// TwinCAT 3 PLC project PLC1
// Title: TcHAL
// Company: none
// Author: Tobias Freyermuth
// ProjectVersion: 0.1.4
// Description: Hardware Abstraction Layer of TwinCAT fieldbus devices
// ProgramVersion: 3.1.4024.12
// libraries:
//   Tc2_EtherCAT, * (Beckhoff Automation GmbH)
//   Tc2_Standard, * (Beckhoff Automation GmbH)
//   Tc2_System, * (Beckhoff Automation GmbH)
//   Tc3_Module, * (Beckhoff Automation GmbH)
//   TcUnit, * (www.tcunit.org)
// project tree:
//   analog_input/temperature/ EL3202_0010.TcPOU
//   analog_input/voltage/ EL3164.TcPOU
//   analog_input/_internal/ AI_Voltage_Channel.TcPOU, AI_Temperature_Channel.TcPOU, I_AI_percentage.TcIO, I_AI_Temperature.TcIO, I_AI_Voltage.TcIO
//   analog_output/voltage/ EL4002.TcPOU, EL4102.TcPOU, EL4004.TcPOU, EL4134.TcPOU
//   analog_output/_internal/ AO_Voltage_Channel.TcPOU, I_AO_percentage.TcIO, I_AO_Voltage.TcIO
//   coupler/ EK1101.TcPOU
//   digital_input/ EL1008.TcPOU, EL1104.TcPOU, EL1144.TcPOU, EL1808.TcPOU, EL1124.TcPOU, EL1809.TcPOU
//   digital_input/_internal/ HAL_DI_Channel.TcPOU, I_HAL_DI.TcIO
//   digital_output/ EL2008.TcPOU, EL2124.TcPOU, EL2024_0010.TcPOU, EL2502.TcPOU (excluded from build), EL2595.TcPOU, EL2612.TcPOU, EL2521.TcPOU (excluded from build), EL2004.TcPOU, EL2634.TcPOU, EL2808.TcPOU, EL2624.TcPOU, EL2794.TcPOU
//   digital_output/_internal/ HAL_DO_Channel.TcPOU, I_HAL_DO.TcIO
//   / HAL_ErrorEnum.TcDUT, MAIN.TcPOU, PlcTask.TcTTO, Settings.TcGVL, _internal.TcGVL
//   InterfaceManager/ InterfaceManager.TcPOU, InterfaceManager_test.TcPOU, I_AI_Percentage_register.TcDUT, I_AO_Percentage_register.TcDUT, I_AO_Voltage_register.TcDUT, I_AI_Voltage_register.TcDUT, I_InterfaceManager.TcIO
//   Project Information/ F_GetCompany.TcPOU, F_GetTitle.TcPOU (not stored), F_GetVersion.TcPOU
//   Version/ Global_Version.TcGVL
//   _internal/CoE/BeckhoffTerminalConfigEnums/ ENU_DT0800EN02.TcDUT (not stored), ENU_DT0801EN03.TcDUT (not stored)
//   _internal/CoE/buffer/ ring_buffer_CoE_read.TcPOU
//   _internal/CoE/ CoE_buffer_type_cast_union.TcDUT (not stored), CoE_communication_handler.TcPOU, CoE_property_handler.TcPOU, CoE_UML_Class Diagram.TcCD (not stored), I_CoE_config_common.TcIO, I_CoE_property.TcIO, I_CoE_communication_handler.TcIO
//   _internal/CoE/properties/ CoE_property.TcPOU, CoE_property_bool.TcPOU, CoE_property_dint.TcPOU, CoE_property_int.TcPOU, CoE_property_string.TcPOU, CoE_property_udint.TcPOU, CoE_property_uint.TcPOU, CoE_property_usint.TcPOU
//   _internal/ I_device_control.TcIO, I_terminal_channel.TcIO, I_coupler_execution.TcIO, I_terminal_execution.TcIO, linear_adc_to_phy.TcPOU, linear_phy_to_adc.TcPOU, linear_phy_to_adc_test.TcPOU, linear_adc_to_phy_test.TcPOU
// real-time tasks:
//   TASK PlcTask: cycle T#10ms, priority 20, ADS port 350

CONFIGURATION PLC1
    RESOURCE PLC ON TwinCAT3
        TASK PlcTask(INTERVAL := T#10ms, PRIORITY := 20);
        PROGRAM MAIN WITH PlcTask : MAIN;
    END_RESOURCE
END_CONFIGURATION

// ---- HAL_ErrorEnum.TcDUT
(**
This error enum is the central error return type used accross all POUs within TcHAL.
*)

{attribute 'qualified_only'}
{attribute 'strict'}
TYPE HAL_ErrorEnum :
(
	no_error := 0,
	// Error messages related to InterfaceManager
	terminal_not_found, 
	interface_can_not_be_null,
	terminal_name_can_not_be_empty,
	channel_number_out_of_range,
	device_id_can_not_be_null,
	no_empty_space_found_in_register,
	requested_interface_not_found,
	interface_already_in_use,
	max_registration_limit_per_cycle_reached,
    physical_value_too_big,
    physical_value_too_small,
    dx_zero_or_smaller,
    m_zero_or_smaller
);
END_TYPE

// ---- InterfaceManager/I_AI_Percentage_register.TcDUT
TYPE I_AI_Percentage_register :
STRUCT
	registered_interface			: I_AI_Percentage;
	terminal_id 					: UINT;
	channel_number 					: USINT;
	connected_device_id				: UINT;
END_STRUCT
END_TYPE

// ---- InterfaceManager/I_AO_Percentage_register.TcDUT
TYPE I_AO_Percentage_register :
STRUCT
	registered_interface			: I_AO_Percentage;
	terminal_id 					: UINT;
	channel_number 					: USINT;
	connected_device_id				: UINT;
END_STRUCT
END_TYPE

// ---- InterfaceManager/I_AO_Voltage_register.TcDUT
TYPE I_AO_Voltage_register :
STRUCT
	registered_interface			: I_AO_Voltage;
	terminal_id 					: UINT;
	channel_number 					: USINT;
	connected_device_id				: UINT;
END_STRUCT
END_TYPE

// ---- InterfaceManager/I_AI_Voltage_register.TcDUT
TYPE I_AI_Voltage_register :
STRUCT
	registered_interface			: I_AI_Voltage;
	terminal_id 					: UINT;
	channel_number 					: USINT;
	connected_device_id				: UINT;
END_STRUCT
END_TYPE

// ---- Settings.TcGVL
VAR_GLOBAL CONSTANT
	NUMBER_OF_TERMINALS 	: UINT:=200;

	NUMBER_OF_I_HAL_AO_Voltage_INTERFACES		: UINT:=10;
	NUMBER_OF_I_HAL_AI_Voltage_INTERFACES		: UINT:=10;
	NUMBER_OF_I_AI_Percentage_INTERFACES		: UINT:=10;

END_VAR

// ---- Version/Global_Version.TcGVL
{attribute 'TcGenerated'}
{attribute 'no-analysis'}
{attribute 'linkalways'}
// This function has been automatically generated from the project information.
VAR_GLOBAL CONSTANT
	{attribute 'const_non_replaced'}
	stLibVersion_TcHAL : ST_LibVersion := (iMajor := 0, iMinor := 1, iBuild := 4, iRevision := 0, nFlags := 0, sVersion := '0.1.4');
END_VAR

// ---- _internal.TcGVL
{attribute 'qualified_only'}
VAR_GLOBAL
	InterfaceManager_InstanceCounter :UINT;
END_VAR

// ---- analog_input/_internal/I_AI_percentage.TcIO
INTERFACE I_AI_percentage

PROPERTY max_value : real
GET
END_GET
SET
END_SET
END_PROPERTY

PROPERTY min_value : real
GET
END_GET
SET
END_SET
END_PROPERTY

PROPERTY value : real
GET
END_GET
END_PROPERTY

END_INTERFACE

// ---- analog_input/_internal/I_AI_Temperature.TcIO
INTERFACE I_AI_Temperature

PROPERTY errId : HAL_ErrorEnum
GET
END_GET
END_PROPERTY

PROPERTY value : real
GET
END_GET
END_PROPERTY

END_INTERFACE

// ---- analog_input/_internal/I_AI_Voltage.TcIO
INTERFACE I_AI_Voltage

PROPERTY errId : HAL_ErrorEnum
GET
END_GET
END_PROPERTY

PROPERTY rValue : real
GET
END_GET
END_PROPERTY

END_INTERFACE

// ---- analog_output/_internal/I_AO_percentage.TcIO
INTERFACE I_AO_percentage

PROPERTY max_value : real
GET
END_GET
SET
END_SET
END_PROPERTY

PROPERTY min_value : real
GET
END_GET
SET
END_SET
END_PROPERTY

PROPERTY value : real
GET
END_GET
END_PROPERTY

END_INTERFACE

// ---- analog_output/_internal/I_AO_Voltage.TcIO
INTERFACE I_AO_Voltage

PROPERTY errId : HAL_ErrorEnum
GET
END_GET
END_PROPERTY

PROPERTY rValue : real
GET
END_GET
SET
END_SET
END_PROPERTY

END_INTERFACE

// ---- digital_input/_internal/I_HAL_DI.TcIO
INTERFACE I_HAL_DI

PROPERTY errId : uint
GET
END_GET
END_PROPERTY

PROPERTY xValue : bool
GET
END_GET
END_PROPERTY

END_INTERFACE

// ---- digital_output/_internal/I_HAL_DO.TcIO
INTERFACE I_HAL_DO

PROPERTY errId : HAL_ErrorEnum
GET
END_GET
END_PROPERTY

PROPERTY xValue : bool
GET
END_GET
SET
END_SET
END_PROPERTY

END_INTERFACE

// ---- InterfaceManager/I_InterfaceManager.TcIO
INTERFACE I_InterfaceManager

METHOD register_I_AI_Percentage : BOOL
VAR_INPUT
	interface_to_be_registered		: I_AI_Percentage;
	terminal_id 					: UINT;
	channel_number 					: USINT; 
END_VAR
VAR_OUTPUT
	errId		: HAL_ErrorEnum;
END_VAR
END_METHOD

METHOD register_I_AI_Temperature : BOOL
VAR_INPUT
	interface_to_be_registered		: I_AI_Temperature;
	terminal_id 					: UINT;
	channel_number 					: USINT; 
END_VAR
VAR_OUTPUT
	errId		: HAL_ErrorEnum;
END_VAR
END_METHOD

METHOD register_I_AI_Voltage : BOOL
VAR_INPUT
	interface_to_be_registered		: I_AI_Voltage;
	terminal_id 					: UINT;
	channel_number 					: USINT; 
END_VAR
VAR_OUTPUT
	errId		: HAL_ErrorEnum;
END_VAR
END_METHOD

METHOD register_I_AO_Percentage : BOOL
VAR_INPUT
	interface_to_be_registered		: I_AO_Percentage;
	terminal_id 					: UINT;
	channel_number 					: USINT; 
END_VAR
VAR_OUTPUT
	errId		: HAL_ErrorEnum;
END_VAR
END_METHOD

METHOD register_I_AO_Voltage : BOOL
VAR_INPUT
	interface_to_be_registered		: I_AO_Voltage;
	terminal_id 					: UINT;
	channel_number 					: USINT; 
END_VAR
VAR_OUTPUT
	errId		: HAL_ErrorEnum;
END_VAR
END_METHOD

METHOD register_terminal : BOOL
VAR_INPUT
	terminal_name : STRING;
END_VAR
VAR_OUTPUT
	errId : HAL_ErrorEnum;
    terminalId : UINT;
END_VAR
END_METHOD

END_INTERFACE

// ---- _internal/CoE/I_CoE_config_common.TcIO
INTERFACE I_CoE_config_common

METHOD get_DeviceName : BOOL
VAR_OUTPUT
	value: STRING;
END_VAR
END_METHOD

METHOD get_DeviceType : BOOL
VAR_OUTPUT
	value: UDINT;
END_VAR
END_METHOD

METHOD get_ProductCode : BOOL
VAR_OUTPUT
	value 	: UDINT; 
END_VAR
END_METHOD

METHOD get_Revision : BOOL
VAR_OUTPUT
	value 	: UDINT; 
END_VAR
END_METHOD

METHOD get_SerialNumber : BOOL
VAR_OUTPUT
	value 	: UDINT; 
END_VAR
END_METHOD

METHOD get_SoftwareVersion : BOOL
VAR_OUTPUT
	value: STRING(2);
END_VAR
END_METHOD

METHOD get_VendorId : BOOL
VAR_OUTPUT
	value: UDINT;
END_VAR
END_METHOD

METHOD getHardwareVersion : BOOL
VAR_OUTPUT
	value: STRING(2);
END_VAR
END_METHOD

END_INTERFACE

// ---- _internal/CoE/I_CoE_property.TcIO
INTERFACE I_CoE_property

PROPERTY CoE_communication_handler : I_CoE_communication_handler
GET
END_GET
SET
END_SET
END_PROPERTY

PROPERTY dataTypeSize : uint
GET
END_GET
END_PROPERTY

METHOD handle_read_callback : BOOL
VAR_INPUT
	pt_buffer : POINTER TO CoE_buffer_type_cast_union;
	errId: UDINT;
END_VAR
END_METHOD

METHOD handle_write_callback : BOOL
VAR_INPUT
	errId : UDINT;
END_VAR
END_METHOD

PROPERTY Index : word
GET
END_GET
END_PROPERTY

PROPERTY init_done : bool
GET
END_GET
END_PROPERTY

(**
This method is initializing or reinitializing the property and returns TRUE when this is done.
In case of an error during the init it returns the ErrorCode related to the error that occurred.
*)
METHOD reinit : BOOL
VAR_OUTPUT
	errId: UDINT;
END_VAR
END_METHOD

METHOD run : BOOL
VAR_INPUT
END_VAR
END_METHOD

PROPERTY SlaveAddress : UINT
GET
END_GET
SET
END_SET
END_PROPERTY

PROPERTY SubIndex : BYTE
GET
END_GET
END_PROPERTY

PROPERTY valueToWrite : CoE_buffer_type_cast_union
GET
END_GET
END_PROPERTY

END_INTERFACE

// ---- _internal/CoE/I_CoE_communication_handler.TcIO
INTERFACE I_CoE_communication_handler

METHOD add_read_request : BOOL
VAR_INPUT
	request	: I_CoE_property;
END_VAR
END_METHOD

METHOD add_write_request : BOOL
VAR_INPUT
	request	: I_CoE_property;
END_VAR
END_METHOD

END_INTERFACE

// ---- _internal/I_device_control.TcIO
INTERFACE I_device_control

METHOD release_control : BOOL
VAR_INPUT
	device_id : DWORD;
END_VAR
END_METHOD

METHOD request_control : BOOL
VAR_INPUT
	device_id : DWORD;
END_VAR
END_METHOD

END_INTERFACE

// ---- _internal/I_terminal_channel.TcIO
INTERFACE I_terminal_channel

METHOD register_channel : BOOL
VAR_INPUT
    terminalId : UINT;
    I_interface_manager : I_interfaceManager;
END_VAR
VAR_OUTPUT
	errId		: HAL_ErrorEnum;
END_VAR
END_METHOD

END_INTERFACE

// ---- _internal/I_coupler_execution.TcIO
INTERFACE I_coupler_execution

METHOD run : BOOL
VAR_INPUT
	sync_unit_ok : BOOL;
END_VAR
END_METHOD

END_INTERFACE

// ---- _internal/I_terminal_execution.TcIO
INTERFACE I_terminal_execution

METHOD run : BOOL
VAR_INPUT
END_VAR
END_METHOD

END_INTERFACE

// ---- MAIN.TcPOU
PROGRAM MAIN
VAR
	linear_phy_to_adc_test_ 		: linear_phy_to_adc_test;
	linear_adc_to_phy_test_ 		: linear_adc_to_phy_test;
	InterfaceManager_test_ 			: InterfaceManager_test;
	
	coe_handler : CoE_communication_handler;
	interface_manager :InterfaceManager;

	// Terminal_1 : EK1101
	Terminal_2 : EL1808(CoE_communication_handler:=coe_handler );
	Terminal_3 : EL2808(CoE_communication_handler:=coe_handler );
	Terminal_4 : EL4002(CoE_communication_handler:=coe_handler, InterfaceManager:=interface_manager, name:='Terminal_4');
	// Terminal_5 : 
	Terminal_6 : EL3164(CoE_communication_handler:=coe_handler, InterfaceManager:=interface_manager, name:='Terminal_6');
	// Terminal_7 :

END_VAR

TcUnit.RUN();

END_PROGRAM

// ---- _internal/linear_phy_to_adc_test.TcPOU
FUNCTION_BLOCK INTERNAL linear_phy_to_adc_test EXTENDS TcUnit.FB_TestSuite
VAR_INPUT
END_VAR
VAR_OUTPUT
END_VAR
VAR
END_VAR

test_physical_values_out_of_range();
test_typical_setting_and_values_0_to_10();
test_typical_setting_and_values_4_to_20();  // ToDo, this needs to be verified with real hardware 
test_typical_setting_and_values_minus_10_to_10();
test_zero_adc_min_and_max();
test_zero_physical_min_and_max();

METHOD test_physical_values_out_of_range
VAR_INPUT
END_VAR
VAR
		returned_result			: BOOL;
		returned_adc_value		: DINT;
		returned_errId 			: HAL_ErrorEnum;
		
		// call function with physical value = 12.9
		case_1_expected_result  		: BOOL:=FALSE;
		case_1_expected_adc_value		: DINT;
		case_1_expected_errId 			: UINT:=1;
		
		// call function with physical value = -12.9
		case_2_expected_result  		: BOOL:=FALSE;
		case_2_expected_adc_value		: DINT;
		case_2_expected_errId 			: UINT:=2;

END_VAR
TEST('test_physical_values_out_of_range');


// ======================================
// Test case 1, 
// call with physical value 12.9
// ====
returned_result:=linear_phy_to_adc(physical_min:=-10 , physical_max:=10 , adc_min:=-32767 , adc_max:=32767 , physical_value:=12.9 , adc_value=>returned_adc_value , errId=>returned_errId );

AssertEquals(Expected := case_1_expected_result,
             Actual := returned_result,
             Message := 'Fucntion returns incorrect result,');
			 
AssertEquals(Expected := case_1_expected_adc_value,
             Actual := returned_adc_value,
             Message := 'Fucntion returns incorrect adc_value,');		 

AssertEquals(Expected :=case_1_expected_errId ,
             Actual := returned_errId ,
             Message := 'Fucntion returns incorrect errId,');
			 
			 
// ======================================
// Test case 2, 
// call with physical value -12.9
// ====
returned_result:=linear_phy_to_adc(physical_min:=-10 , physical_max:=10 , adc_min:=-32767 , adc_max:=32767 , physical_value:=-12.9 , adc_value=>returned_adc_value , errId=>returned_errId );

AssertEquals(Expected := case_2_expected_result,
             Actual := returned_result,
             Message := 'Fucntion returns incorrect result,');
			 
AssertEquals(Expected := case_2_expected_adc_value,
             Actual := returned_adc_value,
             Message := 'Fucntion returns incorrect adc_value,');		 

AssertEquals(Expected :=case_2_expected_errId ,
             Actual := returned_errId ,
             Message := 'Fucntion returns incorrect errId,');
			 
			 
		 
			 
TEST_FINISHED();
END_METHOD

METHOD test_typical_setting_and_values_0_to_10
VAR_INPUT
END_VAR
VAR
		returned_result			: BOOL;
		returned_adc_value		: DINT;
		returned_errId 			: HAL_ErrorEnum;
		
		// call function with physical value = 0
		case_1_physical_value			: REAL:=0.0;
		case_1_expected_result  		: BOOL:=TRUE;
		case_1_expected_adc_value		: DINT:=0;
		case_1_expected_errId 			: UINT:=0;
		
		// call with physical value somewhere in the middle of its range
		case_2_physical_value			: REAL:=4.95;
		case_2_expected_result  		: BOOL:=TRUE;
		case_2_expected_adc_value		: DINT:=16220;
		case_2_expected_errId 			: UINT:=0;
		
		// ccall with physical max value
		case_3_physical_value			: REAL:=10.0;
		case_3_expected_result  		: BOOL:=TRUE;
		case_3_expected_adc_value		: DINT:=32767;
		case_3_expected_errId 			: UINT:=0;
END_VAR
TEST('test_typical_setting_and_values_0_to_10');


// ======================================
// Test case 1
// call with physical min value
// ====
returned_result:=linear_phy_to_adc(physical_min:=0 , physical_max:=10 , adc_min:=0 , adc_max:=32767 , physical_value:=case_1_physical_value , adc_value=>returned_adc_value , errId=>returned_errId );

AssertEquals(Expected := case_1_expected_result,
             Actual := returned_result,
             Message := 'Test case 1 fucntion returns incorrect result,');
			 
AssertEquals(Expected := case_1_expected_adc_value,
             Actual := returned_adc_value,
             Message := 'Test case 1 fucntion returns incorrect adc_value,');		 

AssertEquals(Expected :=case_1_expected_errId ,
             Actual := returned_errId ,
             Message := 'Test case 1 fucntion returns incorrect errId,');


// ======================================
// Test case 2, 
// call with physical value somewhere in the middle of its range
// ====
returned_result:=linear_phy_to_adc(physical_min:=0 , physical_max:=10 , adc_min:=0 , adc_max:=32767 , physical_value:=case_2_physical_value , adc_value=>returned_adc_value , errId=>returned_errId );

AssertEquals(Expected := case_2_expected_result,
             Actual := returned_result,
             Message := 'Test case 2 fcntion returns incorrect result,');
			 
AssertEquals(Expected := case_2_expected_adc_value,
             Actual := returned_adc_value,
             Message := 'Test case 2 fucntion returns incorrect adc_value,');		 

AssertEquals(Expected :=case_2_expected_errId ,
             Actual := returned_errId ,
             Message := 'Test case 2 fucntion returns incorrect errId,');


// ======================================
// Test case 3,
// call with physical max value
// ====
returned_result:=linear_phy_to_adc(physical_min:=0 , physical_max:=10 , adc_min:=0 , adc_max:=32767 , physical_value:=case_3_physical_value , adc_value=>returned_adc_value , errId=>returned_errId );

AssertEquals(Expected := case_3_expected_result,
             Actual := returned_result,
             Message := 'Test case 3 fucntion returns incorrect result,');
			 
AssertEquals(Expected := case_3_expected_adc_value,
             Actual := returned_adc_value,
             Message := 'Test case 3 fucntion returns incorrect adc_value,');		 

AssertEquals(Expected :=case_3_expected_errId ,
             Actual := returned_errId ,
             Message := 'Test case 3 fucntion returns incorrect errId,');			 
			 
			 
TEST_FINISHED();
END_METHOD

METHOD test_typical_setting_and_values_4_to_20
VAR_INPUT
END_VAR
VAR
		returned_result			: BOOL;
		returned_adc_value		: DINT;
		returned_errId 			: HAL_ErrorEnum;
		
		// call with physical min value
		case_1_physical_value			: REAL:=0.0;
		case_1_expected_result  		: BOOL:=TRUE;
		case_1_expected_adc_value		: DINT:=0;
		case_1_expected_errId 			: UINT:=0;
		
		// call with physical value somewhere in the middle of its range
		case_2_physical_value			: REAL:=9.95;
		case_2_expected_result  		: BOOL:=TRUE;
		case_2_expected_adc_value		: DINT:=16302;
		case_2_expected_errId 			: UINT:=0;
		
		// call with physical max value
		case_3_physical_value			: REAL:=20.0;
		case_3_expected_result  		: BOOL:=TRUE;
		case_3_expected_adc_value		: DINT:=32767;
		case_3_expected_errId 			: UINT:=0;
END_VAR
TEST('test_typical_setting_and_values_4_to_20');


// ======================================
// Test case 1
// call with physical min value
// ====
returned_result:=linear_phy_to_adc(physical_min:=0 , physical_max:=20 , adc_min:=0 , adc_max:=32767 , physical_value:=case_1_physical_value , adc_value=>returned_adc_value , errId=>returned_errId );

AssertEquals(Expected := case_1_expected_result,
             Actual := returned_result,
             Message := 'Test case 1 fucntion returns incorrect result,');
			 
AssertEquals(Expected := case_1_expected_adc_value,
             Actual := returned_adc_value,
             Message := 'Test case 1 fucntion returns incorrect adc_value,');		 

AssertEquals(Expected :=case_1_expected_errId ,
             Actual := returned_errId ,
             Message := 'Test case 1 fucntion returns incorrect errId,');


// ======================================
// Test case 2,
// call with physical value somewhere in the middle of its range
// ====
returned_result:=linear_phy_to_adc(physical_min:=0 , physical_max:=20 , adc_min:=0 , adc_max:=32767 , physical_value:=case_2_physical_value , adc_value=>returned_adc_value , errId=>returned_errId );

AssertEquals(Expected := case_2_expected_result,
             Actual := returned_result,
             Message := 'Test case 2 fcntion returns incorrect result,');
			 
AssertEquals(Expected := case_2_expected_adc_value,
             Actual := returned_adc_value,
             Message := 'Test case 2 fucntion returns incorrect adc_value,');		 

AssertEquals(Expected :=case_2_expected_errId ,
             Actual := returned_errId ,
             Message := 'Test case 2 fucntion returns incorrect errId,');


// ======================================
// Test case 3,
// call with physical max value
// ====
returned_result:=linear_phy_to_adc(physical_min:=0 , physical_max:=20 , adc_min:=0 , adc_max:=32767 , physical_value:=case_3_physical_value , adc_value=>returned_adc_value , errId=>returned_errId );

AssertEquals(Expected := case_3_expected_result,
             Actual := returned_result,
             Message := 'Test case 3 fucntion returns incorrect result,');
			 
AssertEquals(Expected := case_3_expected_adc_value,
             Actual := returned_adc_value,
             Message := 'Test case 3 fucntion returns incorrect adc_value,');		 

AssertEquals(Expected :=case_3_expected_errId ,
             Actual := returned_errId ,
             Message := 'Test case 3 fucntion returns incorrect errId,');			 
			 
			 
TEST_FINISHED();
END_METHOD

METHOD test_typical_setting_and_values_minus_10_to_10
VAR_INPUT
END_VAR
VAR
		returned_result			: BOOL;
		returned_adc_value		: INT;
		returned_errId 			: HAL_ErrorEnum;
		
		// call with physical value 0
		case_1_physical_value			: REAL:=0.0;
		case_1_expected_result  		: BOOL:=TRUE;
		case_1_expected_adc_value		: INT:=0;
		case_1_expected_errId 			: UINT:=0;
		
		// call with physical min value
		case_2_physical_value			: REAL:=-10.0;
		case_2_expected_result  		: BOOL:=TRUE;
		case_2_expected_adc_value		: INT:=-32767;
		case_2_expected_errId 			: UINT:=0;
		
		// call with physical max value
		case_3_physical_value			: REAL:=10.0;
		case_3_expected_result  		: BOOL:=TRUE;
		case_3_expected_adc_value		: INT:=32767;
		case_3_expected_errId 			: UINT:=0;
		
		// call with physical value somewhere in the middle of its range
		case_4_physical_value			: REAL:=4.95;
		case_4_expected_result  		: BOOL:=TRUE;
		case_4_expected_adc_value		: INT:=16220;
		case_4_expected_errId 			: UINT:=0;
END_VAR
TEST('test_typical_setting_and_values_minus_10_to_10');


// ======================================
// Test case 1, 
// call with physical value 0
// ====
returned_result:=linear_phy_to_adc(physical_min:=-10 , physical_max:=10 , adc_min:=-32767 , adc_max:=32767 , physical_value:=case_1_physical_value , adc_value=>returned_adc_value , errId=>returned_errId );

AssertEquals(Expected := case_1_expected_result,
             Actual := returned_result,
             Message := 'Test case 1 fucntion returns incorrect result,');
			 
AssertEquals(Expected := case_1_expected_adc_value,
             Actual := returned_adc_value,
             Message := 'Test case 1 fucntion returns incorrect adc_value,');		 

AssertEquals(Expected :=case_1_expected_errId ,
             Actual := returned_errId ,
             Message := 'Test case 1 fucntion returns incorrect errId,');


// ======================================
// Test case 2, 
// call with physical min value
// ====
returned_result:=linear_phy_to_adc(physical_min:=-10 , physical_max:=10 , adc_min:=-32767 , adc_max:=32767 , physical_value:=case_2_physical_value , adc_value=>returned_adc_value , errId=>returned_errId );

AssertEquals(Expected := case_2_expected_result,
             Actual := returned_result,
             Message := 'Test case 2 fcntion returns incorrect result,');
			 
AssertEquals(Expected := case_2_expected_adc_value,
             Actual := returned_adc_value,
             Message := 'Test case 2 fucntion returns incorrect adc_value,');		 

AssertEquals(Expected :=case_2_expected_errId ,
             Actual := returned_errId ,
             Message := 'Test case 2 fucntion returns incorrect errId,');


// ======================================
// Test case 3,
// call with physical max value
// ====
returned_result:=linear_phy_to_adc(physical_min:=-10 , physical_max:=10 , adc_min:=-32767 , adc_max:=32767 , physical_value:=case_3_physical_value , adc_value=>returned_adc_value , errId=>returned_errId );

AssertEquals(Expected := case_3_expected_result,
             Actual := returned_result,
             Message := 'Test case 3 fucntion returns incorrect result,');
			 
AssertEquals(Expected := case_3_expected_adc_value,
             Actual := returned_adc_value,
             Message := 'Test case 3 fucntion returns incorrect adc_value,');		 

AssertEquals(Expected :=case_3_expected_errId ,
             Actual := returned_errId ,
             Message := 'Test case 3 fucntion returns incorrect errId,');			 

// ======================================
// Test case 4,
// call with physical value somewhere in the middle of its range
// ====
returned_result:=linear_phy_to_adc(physical_min:=-10 , physical_max:=10 , adc_min:=-32767 , adc_max:=32767 , physical_value:=case_4_physical_value , adc_value=>returned_adc_value , errId=>returned_errId );

AssertEquals(Expected := case_4_expected_result,
             Actual := returned_result,
             Message := 'Test case 4 fucntion returns incorrect result,');
			 
AssertEquals(Expected := case_4_expected_adc_value,
             Actual := returned_adc_value,
             Message := 'Test case 4 fucntion returns incorrect adc_value,');		 

AssertEquals(Expected :=case_4_expected_errId ,
             Actual := returned_errId ,
             Message := 'Test case 4 fucntion returns incorrect errId,');	 
			 
TEST_FINISHED();
END_METHOD

METHOD test_zero_adc_min_and_max
VAR_INPUT
END_VAR
VAR
		returned_result			: BOOL;
		returned_adc_value		: DINT;
		returned_errId 			: HAL_ErrorEnum;
		
		// call function with physical value = 0
		case_1_expected_result  		: BOOL:=FALSE;
		case_1_expected_adc_value		: DINT;
		case_1_expected_errId 			: UINT:=3;
		
		// call function with physical value = 5.5
		case_2_expected_result  		: BOOL:=FALSE;
		case_2_expected_adc_value		: DINT;
		case_2_expected_errId 			: UINT:=3;
		
		// call function with physical value = -5.5
		case_3_expected_result  		: BOOL:=FALSE;
		case_3_expected_adc_value		: DINT;
		case_3_expected_errId 			: UINT:=2;
END_VAR
TEST('test_zero_adc_min_and_max');


// ======================================
// Test case 1, 
// call with physical value 0
// ====
returned_result:=linear_phy_to_adc(physical_min:=0 , physical_max:=10 , adc_min:=0 , adc_max:=0 , physical_value:=0 , adc_value=>returned_adc_value , errId=>returned_errId );

AssertEquals(Expected := case_1_expected_result,
             Actual := returned_result,
             Message := 'Fucntion returns incorrect result,');
			 
AssertEquals(Expected := case_1_expected_adc_value,
             Actual := returned_adc_value,
             Message := 'Fucntion returns incorrect adc_value,');		 

AssertEquals(Expected :=case_1_expected_errId ,
             Actual := returned_errId ,
             Message := 'Fucntion returns incorrect errId,');
			 
			 
// ======================================
// Test case 2, 
// call with physical value 5.5
// ====
returned_result:=linear_phy_to_adc(physical_min:=0 , physical_max:=10 , adc_min:=0 , adc_max:=0 , physical_value:=5.5 , adc_value=>returned_adc_value , errId=>returned_errId );

AssertEquals(Expected := case_2_expected_result,
             Actual := returned_result,
             Message := 'Fucntion returns incorrect result,');
			 
AssertEquals(Expected := case_2_expected_adc_value,
             Actual := returned_adc_value,
             Message := 'Fucntion returns incorrect adc_value,');		 

AssertEquals(Expected :=case_2_expected_errId ,
             Actual := returned_errId ,
             Message := 'Fucntion returns incorrect errId,');
			 
			 
// ======================================
// Test case 1, 
// call with physical value 0
// ====
returned_result:=linear_phy_to_adc(physical_min:=0 , physical_max:=10 , adc_min:=0 , adc_max:=0 , physical_value:=-5.5 , adc_value=>returned_adc_value , errId=>returned_errId );

AssertEquals(Expected := case_3_expected_result,
             Actual := returned_result,
             Message := 'Fucntion returns incorrect result,');
			 
AssertEquals(Expected := case_3_expected_adc_value,
             Actual := returned_adc_value,
             Message := 'Fucntion returns incorrect adc_value,');		 

AssertEquals(Expected :=case_3_expected_errId ,
             Actual := returned_errId ,
             Message := 'Fucntion returns incorrect errId,');
		 
			 
			 
TEST_FINISHED();
END_METHOD

METHOD test_zero_physical_min_and_max
VAR_INPUT
END_VAR
VAR
		returned_result			: BOOL;
		returned_adc_value		: DINT;
		returned_errId 			: HAL_ErrorEnum;
		
		// call function with physical value = 0
		case_1_expected_result  		: BOOL:=FALSE;
		case_1_expected_adc_value		: DINT;
		case_1_expected_errId 			: UINT:=4;
		
		// call function with physical value = 5.5
		case_2_expected_result  		: BOOL:=FALSE;
		case_2_expected_adc_value		: DINT;
		case_2_expected_errId 			: UINT:=1;
		
		// call function with physical value = -5.5
		case_3_expected_result  		: BOOL:=FALSE;
		case_3_expected_adc_value		: DINT;
		case_3_expected_errId 			: UINT:=2;
END_VAR
TEST('test_zero_physical_min_and_or_max');


// ======================================
// Test case 1, 
// call with physical value 0
// ====
returned_result:=linear_phy_to_adc(physical_min:=0 , physical_max:=0 , adc_min:=0 , adc_max:=32767 , physical_value:=0 , adc_value=>returned_adc_value , errId=>returned_errId );

AssertEquals(Expected := case_1_expected_result,
             Actual := returned_result,
             Message := 'Fucntion returns incorrect result,');
			 
AssertEquals(Expected := case_1_expected_adc_value,
             Actual := returned_adc_value,
             Message := 'Fucntion returns incorrect adc_value,');		 

AssertEquals(Expected :=case_1_expected_errId ,
             Actual := returned_errId ,
             Message := 'Fucntion returns incorrect errId,');
			 
			 
// ======================================
// Test case 2, 
// call with physical value 5.5
// ====
returned_result:=linear_phy_to_adc(physical_min:=0 , physical_max:=0 , adc_min:=0 , adc_max:=32767 , physical_value:=5.5 , adc_value=>returned_adc_value , errId=>returned_errId );

AssertEquals(Expected := case_2_expected_result,
             Actual := returned_result,
             Message := 'Fucntion returns incorrect result,');
			 
AssertEquals(Expected := case_2_expected_adc_value,
             Actual := returned_adc_value,
             Message := 'Fucntion returns incorrect adc_value,');		 

AssertEquals(Expected :=case_2_expected_errId ,
             Actual := returned_errId ,
             Message := 'Fucntion returns incorrect errId,');
			 
			 
// ======================================
// Test case 1, 
// call with physical value 0
// ====
returned_result:=linear_phy_to_adc(physical_min:=0 , physical_max:=0 , adc_min:=0 , adc_max:=32767 , physical_value:=-5.5 , adc_value=>returned_adc_value , errId=>returned_errId );

AssertEquals(Expected := case_3_expected_result,
             Actual := returned_result,
             Message := 'Fucntion returns incorrect result,');
			 
AssertEquals(Expected := case_3_expected_adc_value,
             Actual := returned_adc_value,
             Message := 'Fucntion returns incorrect adc_value,');		 

AssertEquals(Expected :=case_3_expected_errId ,
             Actual := returned_errId ,
             Message := 'Fucntion returns incorrect errId,');
		 
			 
			 
TEST_FINISHED();
END_METHOD

END_FUNCTION_BLOCK

// ---- _internal/linear_phy_to_adc.TcPOU
(**
This function is sacling a physical value to a adc value with 

*)
FUNCTION linear_phy_to_adc : BOOL
VAR_INPUT
	physical_min : INT;
	physical_max : INT;
	adc_min : INT;
	adc_max : INT;
	physical_value : REAL;
END_VAR
VAR_OUTPUT
	adc_value : INT;
	errId 	  : HAL_ErrorEnum;
END_VAR
VAR
	dx: DINT;
	dy: DINT;
    
	m: REAL;
	b: REAL;
END_VAR


IF physical_value > INT_TO_REAL(physical_max) THEN
	linear_phy_to_adc:=FALSE;
	errId := HAL_ErrorEnum.physical_value_too_big;
ELSIF physical_value < INT_TO_REAL(physical_min) THEN 
	linear_phy_to_adc:=FALSE;
	errId := HAL_ErrorEnum.physical_value_too_small;
ELSE
	dx := adc_max - adc_min;
	dy := physical_max - physical_min;
	IF dx <= 0 THEN
		linear_phy_to_adc:=FALSE;
		errId := HAL_ErrorEnum.dx_zero_or_smaller;
	ELSE
		m := DINT_TO_REAL(dy) / DINT_TO_REAL(dx);
		IF m <= 0 THEN
			linear_phy_to_adc:=FALSE;
			errId := HAL_ErrorEnum.m_zero_or_smaller;
		ELSE
			b := INT_TO_REAL(physical_min) - m * INT_TO_REAL(adc_min);
			adc_value := REAL_TO_INT(physical_value/m - b/m);
			linear_phy_to_adc:=TRUE;
		END_IF
	END_IF
END_IF

END_FUNCTION

// ---- _internal/linear_adc_to_phy_test.TcPOU
FUNCTION_BLOCK INTERNAL linear_adc_to_phy_test EXTENDS TcUnit.FB_TestSuite
VAR_INPUT
END_VAR
VAR_OUTPUT
END_VAR
VAR
END_VAR

test_adc_values_out_of_range();
test_typical_setting_and_values_0_to_10();

// test_typical_setting_and_values_4_to_20();  // ToDo, this needs to be verified with real hardware 

test_typical_setting_and_values_minus_10_to_10();
test_zero_phy_min_and_max();
test_zero_adc_min_and_max();

METHOD test_adc_values_out_of_range
VAR_INPUT
END_VAR
VAR
		returned_result			: BOOL;
		returned_phy_value		: REAL;
		returned_errId 			: HAL_ErrorEnum;
		
		// call with adc value 23000
		case_1_expected_result  		: BOOL:=FALSE;
		case_1_expected_adc_value		: REAL;
		case_1_expected_errId 			: UINT:=1;
		
		// call with adc value -23000
		case_2_expected_result  		: BOOL:=FALSE;
		case_2_expected_adc_value		: real;
		case_2_expected_errId 			: UINT:=2;

END_VAR
TEST('test_adc_values_out_of_range');


// ======================================
// Test case 1, 
// call with adc value 23000
// ====
returned_result:= linear_adc_to_phy(physical_min:=-10 , physical_max:=10 , adc_min:=-16383 , adc_max:=16383 , adc_value:=23000 , physical_value=>returned_phy_value , errId=>returned_errId );

AssertEquals(Expected := case_1_expected_result,
             Actual := returned_result,
             Message := 'Test case 1 fucntion returns incorrect result,');
			 
AssertEquals(Expected := case_1_expected_adc_value,
             Actual := returned_phy_value,
             Message := 'Test case 1 fucntion incorrect adc_value,');		 

AssertEquals(Expected :=case_1_expected_errId ,
             Actual := returned_errId ,
             Message := 'Test case 1 fucntion incorrect errId,');
			 
			 
// ======================================
// Test case 2, 
// call with adc value -23000
// ====
returned_result:= linear_adc_to_phy(physical_min:=-10 , physical_max:=10 , adc_min:=-16383 , adc_max:=16383 , adc_value:=-23000 , physical_value=>returned_phy_value , errId=>returned_errId );

AssertEquals(Expected := case_2_expected_result,
             Actual := returned_result,
             Message := 'Test case 2 fucntion returns incorrect result,');
			 
AssertEquals(Expected := case_2_expected_adc_value,
             Actual := returned_phy_value,
             Message := 'Test case 2 fucntion returns incorrect adc_value,');		 

AssertEquals(Expected :=case_2_expected_errId ,
             Actual := returned_errId ,
             Message := 'Test case 2 fucntion returns incorrect errId,');
			 
			 
		 
			 
TEST_FINISHED();
END_METHOD

METHOD test_typical_setting_and_values_0_to_10
VAR_INPUT
END_VAR
VAR
		returned_result			: BOOL;
		returned_phy_value		: REAL;
		returned_errId 			: HAL_ErrorEnum;
		
		// call function with physical value = 0
		case_1_adc_value				: INT:=0;
		case_1_expected_result  		: BOOL:=TRUE;
		case_1_expected_phy_value		: REAL:=0.0;
		case_1_expected_errId 			: UINT:=0;
		
		// call with physical value somewhere in the middle of its range
		case_2_adc_value				: INT:=16220;
		case_2_expected_result  		: BOOL:=TRUE;
		case_2_expected_phy_value		: REAL:=4.95;
		case_2_expected_errId 			: UINT:=0;
		
		// ccall with physical max value
		case_3_adc_value				: INT:=32767;
		case_3_expected_result  		: BOOL:=TRUE;
		case_3_expected_phy_value		: REAL:=10.0;
		case_3_expected_errId 			: UINT:=0;
END_VAR
TEST('test_typical_setting_and_values_0_to_10');


// ======================================
// Test case 1
// call with physical min value
// ====
returned_result:= linear_adc_to_phy(physical_min:=0 , physical_max:=10 , adc_min:=0 , adc_max:=32767 , adc_value:=case_1_adc_value , physical_value=>returned_phy_value , errId=>returned_errId );

AssertEquals(Expected := case_1_expected_result,
             Actual := returned_result,
             Message := 'Test case 1 fucntion returns incorrect result,');
			 
AssertEquals(Expected := case_1_expected_phy_value,
             Actual := returned_phy_value,
             Message := 'Test case 1 fucntion returns incorrect adc_value,');		 

AssertEquals(Expected :=case_1_expected_errId ,
             Actual := returned_errId ,
             Message := 'Test case 1 fucntion returns incorrect errId,');


// ======================================
// Test case 2, 
// call with physical value somewhere in the middle of its range
// ====
returned_result:= linear_adc_to_phy(physical_min:=0 , physical_max:=10 , adc_min:=0 , adc_max:=32767 , adc_value:=case_2_adc_value , physical_value=>returned_phy_value , errId=>returned_errId );

AssertEquals(Expected := case_2_expected_result,
             Actual := returned_result,
             Message := 'Test case 2 fcntion returns incorrect result,');
			 
AssertEquals_REAL(Expected:= case_2_expected_phy_value, 
				  Actual:= returned_phy_value, 
			      Delta:= 0.001, 
				  Message:= 'Test case 2 fucntion returns incorrect adc_value,');		 

AssertEquals(Expected :=case_2_expected_errId ,
             Actual := returned_errId ,
             Message := 'Test case 2 fucntion returns incorrect errId,');


// ======================================
// Test case 3,
// call with physical max value
// ====
returned_result:= linear_adc_to_phy(physical_min:=0 , physical_max:=10 , adc_min:=0 , adc_max:=32767 , adc_value:=case_3_adc_value , physical_value=>returned_phy_value , errId=>returned_errId );

AssertEquals(Expected := case_3_expected_result,
             Actual := returned_result,
             Message := 'Test case 3 fucntion returns incorrect result,');

AssertEquals_REAL(Expected:= case_3_expected_phy_value, 
				  Actual:= returned_phy_value, 
			      Delta:= 0.001, 
				  Message:= 'Test case 3 fucntion returns incorrect adc_value,');	

AssertEquals(Expected :=case_3_expected_errId ,
             Actual := returned_errId ,
             Message := 'Test case 3 fucntion returns incorrect errId,');			 
			 
			 
TEST_FINISHED();
END_METHOD

METHOD test_typical_setting_and_values_4_to_20
VAR_INPUT
END_VAR
VAR
		returned_result			: BOOL;
		returned_adc_value		: DINT;
		returned_errId 			: HAL_ErrorEnum;
		
		// call with physical min value
		case_1_physical_value			: REAL:=0.0;
		case_1_expected_result  		: BOOL:=TRUE;
		case_1_expected_adc_value		: DINT:=0;
		case_1_expected_errId 			: UINT:=0;
		
		// call with physical value somewhere in the middle of its range
		case_2_physical_value			: REAL:=9.95;
		case_2_expected_result  		: BOOL:=TRUE;
		case_2_expected_adc_value		: DINT:=16302;
		case_2_expected_errId 			: UINT:=0;
		
		// call with physical max value
		case_3_physical_value			: REAL:=20.0;
		case_3_expected_result  		: BOOL:=TRUE;
		case_3_expected_adc_value		: DINT:=32767;
		case_3_expected_errId 			: UINT:=0;
END_VAR
TEST('test_typical_setting_and_values_4_to_20');


// ======================================
// Test case 1
// call with physical min value
// ====
returned_result:=linear_phy_to_adc(physical_min:=0 , physical_max:=20 , adc_min:=0 , adc_max:=32767 , physical_value:=case_1_physical_value , adc_value=>returned_adc_value , errId=>returned_errId );

AssertEquals(Expected := case_1_expected_result,
             Actual := returned_result,
             Message := 'Test case 1 fucntion returns incorrect result,');
			 
AssertEquals(Expected := case_1_expected_adc_value,
             Actual := returned_adc_value,
             Message := 'Test case 1 fucntion returns incorrect adc_value,');		 

AssertEquals(Expected :=case_1_expected_errId ,
             Actual := returned_errId ,
             Message := 'Test case 1 fucntion returns incorrect errId,');


// ======================================
// Test case 2,
// call with physical value somewhere in the middle of its range
// ====
returned_result:=linear_phy_to_adc(physical_min:=0 , physical_max:=20 , adc_min:=0 , adc_max:=32767 , physical_value:=case_2_physical_value , adc_value=>returned_adc_value , errId=>returned_errId );

AssertEquals(Expected := case_2_expected_result,
             Actual := returned_result,
             Message := 'Test case 2 fcntion returns incorrect result,');
			 
AssertEquals(Expected := case_2_expected_adc_value,
             Actual := returned_adc_value,
             Message := 'Test case 2 fucntion returns incorrect adc_value,');		 

AssertEquals(Expected :=case_2_expected_errId ,
             Actual := returned_errId ,
             Message := 'Test case 2 fucntion returns incorrect errId,');


// ======================================
// Test case 3,
// call with physical max value
// ====
returned_result:=linear_phy_to_adc(physical_min:=0 , physical_max:=20 , adc_min:=0 , adc_max:=32767 , physical_value:=case_3_physical_value , adc_value=>returned_adc_value , errId=>returned_errId );

AssertEquals(Expected := case_3_expected_result,
             Actual := returned_result,
             Message := 'Test case 3 fucntion returns incorrect result,');
			 
AssertEquals(Expected := case_3_expected_adc_value,
             Actual := returned_adc_value,
             Message := 'Test case 3 fucntion returns incorrect adc_value,');		 

AssertEquals(Expected :=case_3_expected_errId ,
             Actual := returned_errId ,
             Message := 'Test case 3 fucntion returns incorrect errId,');			 
			 
			 
TEST_FINISHED();
END_METHOD

METHOD test_typical_setting_and_values_minus_10_to_10
VAR_INPUT
END_VAR
VAR
		returned_result			: BOOL;
		returned_phy_value		: REAL;
		returned_errId 			: HAL_ErrorEnum;
		
		// call with physical value 0
		case_1_adc_value				: INT:=0;
		case_1_expected_result  		: BOOL:=TRUE;
		case_1_expected_phy_value		: REAL:=0.0;
		case_1_expected_errId 			: UINT:=0;
		
		// call with adc min value
		case_2_adc_value				: INT:=-32767;
		case_2_expected_result  		: BOOL:=TRUE;
		case_2_expected_phy_value		: REAL:=-10.0;
		case_2_expected_errId 			: UINT:=0;
		
		// call with adc max value
		case_3_adc_value				: INT:=32767;
		case_3_expected_result  		: BOOL:=TRUE;
		case_3_expected_phy_value		: REAL:=10.0;
		case_3_expected_errId 			: UINT:=0;
		
		// call with physical value somewhere in the middle of its range
		case_4_adc_value				: INT:=16220;
		case_4_expected_result  		: BOOL:=TRUE;
		case_4_expected_phy_value		: REAL:=4.95;
		case_4_expected_errId 			: UINT:=0;
END_VAR
TEST('test_typical_setting_and_values_minus_10_to_10');


// ======================================
// Test case 1, 
// call with adc value 0
// ====
returned_result:= linear_adc_to_phy(physical_min:=-10 , physical_max:=10 , adc_min:=-32767 , adc_max:=32767 , adc_value:=case_1_adc_value , physical_value=>returned_phy_value , errId=>returned_errId );

AssertEquals(Expected := case_1_expected_result,
             Actual := returned_result,
             Message := 'Test case 1 fucntion returns incorrect result,');
			 
AssertEquals(Expected := case_1_expected_phy_value,
             Actual := returned_phy_value,
             Message := 'Test case 1 fucntion returns incorrect adc_value,');		 

AssertEquals(Expected :=case_1_expected_errId ,
             Actual := returned_errId ,
             Message := 'Test case 1 fucntion returns incorrect errId,');


// ======================================
// Test case 2, 
// call with physical min value
// ====
returned_result:= linear_adc_to_phy(physical_min:=-10 , physical_max:=10 , adc_min:=-32767 , adc_max:=32767 , adc_value:=case_2_adc_value , physical_value=>returned_phy_value , errId=>returned_errId );

AssertEquals(Expected := case_2_expected_result,
             Actual := returned_result,
             Message := 'Test case 2 fcntion returns incorrect result,');
			 
AssertEquals(Expected := case_2_expected_phy_value,
             Actual := returned_phy_value,
             Message := 'Test case 2 fucntion returns incorrect adc_value,');		 

AssertEquals(Expected :=case_2_expected_errId ,
             Actual := returned_errId ,
             Message := 'Test case 2 fucntion returns incorrect errId,');


// ======================================
// Test case 3,
// call with physical max value
// ====
returned_result:= linear_adc_to_phy(physical_min:=-10 , physical_max:=10 , adc_min:=-32767 , adc_max:=32767 , adc_value:=case_3_adc_value , physical_value=>returned_phy_value , errId=>returned_errId );

AssertEquals(Expected := case_3_expected_result,
             Actual := returned_result,
             Message := 'Test case 3 fucntion returns incorrect result,');
			 
AssertEquals(Expected := case_3_expected_phy_value,
             Actual := returned_phy_value,
             Message := 'Test case 3 fucntion returns incorrect adc_value,');		 

AssertEquals(Expected :=case_3_expected_errId ,
             Actual := returned_errId ,
             Message := 'Test case 3 fucntion returns incorrect errId,');			 

// ======================================
// Test case 4,
// call with physical value somewhere in the middle of its range
// ====
returned_result:= linear_adc_to_phy(physical_min:=-10 , physical_max:=10 , adc_min:=-32767 , adc_max:=32767 , adc_value:=case_4_adc_value , physical_value=>returned_phy_value , errId=>returned_errId );

AssertEquals(Expected := case_4_expected_result,
             Actual := returned_result,
             Message := 'Test case 4 fucntion returns incorrect result,');
		 
AssertEquals_REAL(Expected:= case_4_expected_phy_value, 
				  Actual:= returned_phy_value, 
			      Delta:= 0.001, 
				  Message:= 'Test case 4 fucntion returns incorrect adc_value,');

AssertEquals(Expected :=case_4_expected_errId ,
             Actual := returned_errId ,
             Message := 'Test case 4 fucntion returns incorrect errId,');	 
			 
TEST_FINISHED();
END_METHOD

METHOD test_zero_adc_min_and_max
VAR_INPUT
END_VAR
VAR
		returned_result			: BOOL;
		returned_phy_value		: REAL;
		returned_errId 			: HAL_ErrorEnum;
		
		// call function with adc value = 0
		case_1_adc_value				: INT:=0;
		case_1_expected_result  		: BOOL:=FALSE;
		case_1_expected_phy_value		: REAL;
		case_1_expected_errId 			: UINT:=4;
		
		// call function with too high adc value 
		case_2_adc_value				: INT:=16220;
		case_2_expected_result  		: BOOL:=FALSE;
		case_2_expected_phy_value		: REAL;
		case_2_expected_errId 			: UINT:=1;
		
		// call function with too low adc value 
		case_3_adc_value				: INT:=-16220;
		case_3_expected_result  		: BOOL:=FALSE;
		case_3_expected_phy_value		: REAL;
		case_3_expected_errId 			: UINT:=2;
END_VAR
TEST('test_zero_adc_min_and_max');


// ======================================
// Test case 1, 
// call with adc value 0
// ====
returned_result:= linear_adc_to_phy(physical_min:=-10 , physical_max:=10 , adc_min:=0 , adc_max:=0 , adc_value:=case_1_adc_value , physical_value=>returned_phy_value , errId=>returned_errId );

AssertEquals(Expected := case_1_expected_result,
             Actual := returned_result,
             Message := 'Test case 1 fucntion returns incorrect result,');
			 
AssertEquals(Expected := case_1_expected_phy_value,
             Actual := returned_phy_value,
             Message := 'Test case 1 fucntion returns incorrect adc_value,');		 

AssertEquals(Expected :=case_1_expected_errId ,
             Actual := returned_errId ,
             Message := 'Test case 1 fucntion returns incorrect errId,');
			 
			 
// ======================================
// Test case 2, 
// call function with too high adc value 
// ====
returned_result:= linear_adc_to_phy(physical_min:=-10 , physical_max:=10 , adc_min:=0 , adc_max:=0 , adc_value:=case_2_adc_value , physical_value=>returned_phy_value , errId=>returned_errId );

AssertEquals(Expected := case_2_expected_result,
             Actual := returned_result,
             Message := 'Test case 2 fucntion returns incorrect result,');
			 
AssertEquals(Expected := case_2_expected_phy_value,
             Actual := returned_phy_value,
             Message := 'Test case 2 fucntion returns incorrect adc_value,');		 

AssertEquals(Expected :=case_2_expected_errId ,
             Actual := returned_errId ,
             Message := 'Test case 2 fucntion returns incorrect errId,');
			 
			 
// ======================================
// Test case 1, 
// call function with too low adc value 
// ====
returned_result:= linear_adc_to_phy(physical_min:=-10 , physical_max:=10 , adc_min:=0 , adc_max:=0 , adc_value:=case_3_adc_value , physical_value=>returned_phy_value , errId=>returned_errId );

AssertEquals(Expected := case_3_expected_result,
             Actual := returned_result,
             Message := 'Test case 3 fucntion returns incorrect result,');
			 
AssertEquals(Expected := case_3_expected_phy_value,
             Actual := returned_phy_value,
             Message := 'Test case 3 fucntion returns incorrect adc_value,');		 

AssertEquals(Expected :=case_3_expected_errId ,
             Actual := returned_errId ,
             Message := 'Test case 3 fucntion returns incorrect errId,');
		 
			 
			 
TEST_FINISHED();
END_METHOD

METHOD test_zero_phy_min_and_max
VAR_INPUT
END_VAR
VAR
		returned_result			: BOOL;
		returned_phy_value		: REAL;
		returned_errId 			: HAL_ErrorEnum;
		
		// call function with adc value = 0
		case_1_adc_value				: INT:=0;
		case_1_expected_result  		: BOOL:=FALSE;
		case_1_expected_phy_value		: REAL;
		case_1_expected_errId 			: UINT:=3;
		
		// call function with too high adc value 
		case_2_adc_value				: INT:=16220;
		case_2_expected_result  		: BOOL:=FALSE;
		case_2_expected_phy_value		: REAL;
		case_2_expected_errId 			: UINT:=3;

END_VAR
TEST('test_zero_phy_min_and_max');


// ======================================
// Test case 1, 
// call with adc value 0
// ====
returned_result:= linear_adc_to_phy(physical_min:=0 , physical_max:=0 , adc_min:=-16383 , adc_max:=16383 , adc_value:=case_1_adc_value , physical_value=>returned_phy_value , errId=>returned_errId );

AssertEquals(Expected := case_1_expected_result,
             Actual := returned_result,
             Message := 'Test case 1 fucntion returns incorrect result,');
			 
AssertEquals(Expected := case_1_expected_phy_value,
             Actual := returned_phy_value,
             Message := 'Test case 1 fucntion returns incorrect adc_value,');		 

AssertEquals(Expected :=case_1_expected_errId ,
             Actual := returned_errId ,
             Message := 'Test case 1 fucntion returns incorrect errId,');
			 
			 
// ======================================
// Test case 2, 
// call function with too high adc value 
// ====
returned_result:= linear_adc_to_phy(physical_min:=0 , physical_max:=0 , adc_min:=-16383 , adc_max:=16383 , adc_value:=case_2_adc_value , physical_value=>returned_phy_value , errId=>returned_errId );

AssertEquals(Expected := case_2_expected_result,
             Actual := returned_result,
             Message := 'Test case 2 fucntion returns incorrect result,');
			 
AssertEquals(Expected := case_2_expected_phy_value,
             Actual := returned_phy_value,
             Message := 'Test case 2 fucntion returns incorrect adc_value,');		 

AssertEquals(Expected :=case_2_expected_errId ,
             Actual := returned_errId ,
             Message := 'Test case 2 fucntion returns incorrect errId,');
			 
TEST_FINISHED();
END_METHOD

END_FUNCTION_BLOCK

// ---- _internal/linear_adc_to_phy.TcPOU

FUNCTION linear_adc_to_phy : BOOL
VAR_INPUT
	physical_min : DINT;
	physical_max : DINT;
	adc_min : DINT;
	adc_max : DINT;
	adc_value : DINT;
END_VAR
VAR_OUTPUT
	physical_value : REAL;
	errId 	: HAL_ErrorEnum;
END_VAR
VAR
	dx: DINT;
	dy: DINT;
    
	m: REAL;
	b: REAL;
END_VAR


IF adc_value > adc_max THEN
	linear_adc_to_phy:=FALSE;
	errId:=1;
ELSIF adc_value < adc_min THEN 
	linear_adc_to_phy:=FALSE;
	errId:=2;
ELSE
	dx := physical_max - physical_min;
	dy := adc_max - adc_min;
	IF dx <= 0 THEN
		linear_adc_to_phy:=FALSE;
		errId:=3;
	ELSE
		m := DINT_TO_REAL(dy) / DINT_TO_REAL(dx);
		IF m <= 0 THEN
			linear_adc_to_phy:=FALSE;
			errId:=4;
		ELSE
			b := DINT_TO_REAL(adc_min) - m * DINT_TO_REAL(physical_min);
			physical_value := DINT_TO_REAL(adc_value)/m - b/m;
			linear_adc_to_phy := TRUE;
		END_IF
	END_IF
END_IF

END_FUNCTION

// ---- InterfaceManager/InterfaceManager_test.TcPOU
FUNCTION_BLOCK InterfaceManager_test EXTENDS TcUnit.FB_TestSuite
VAR_INPUT
END_VAR
VAR_OUTPUT
END_VAR
VAR
END_VAR

test_InitTwice();

METHOD test_InitTwice
VAR_INPUT
END_VAR
VAR 
	fb_1 : InterfaceManager;
//	fb_2 : InterfaceManager;
END_VAR
TEST('test_InitTwice');



TEST_FINISHED();
END_METHOD

END_FUNCTION_BLOCK

// ---- InterfaceManager/InterfaceManager.TcPOU
FUNCTION_BLOCK InterfaceManager IMPLEMENTS I_InterfaceManager
VAR
	registrations_in_cycle 	: UINT;
	terminals : ARRAY[1..NUMBER_OF_Terminals] OF STRING;
	I_AO_Voltage_interfaces 	: ARRAY[0..NUMBER_OF_I_HAL_AO_Voltage_INTERFACES] OF I_AO_Voltage_register;
	I_AI_Voltage_interfaces 	: ARRAY[0..NUMBER_OF_I_HAL_AI_Voltage_INTERFACES] OF I_AI_Voltage_register;
	I_AO_Percentage_interfaces 	: ARRAY[0..NUMBER_OF_I_AI_Percentage_INTERFACES] OF I_AO_Percentage_register;
    I_AI_Percentage_interfaces 	: ARRAY[0..NUMBER_OF_I_AI_Percentage_INTERFACES] OF I_AI_Percentage_register;
END_VAR
VAR CONSTANT 
	MAX_REGISTRATIONS_PER_CYCLE : UINT:=100;
END_VAR

registrations_in_cycle:=0;

METHOD FB_init : BOOL
VAR_INPUT
	bInitRetains : BOOL; // if TRUE, the retain variables are initialized (warm start / cold start)
	bInCopyCode : BOOL;  // if TRUE, the instance afterwards gets moved into the copy code (online change)
END_VAR

VAR
	tmp: UINT;
END_VAR
IF _internal.InterfaceManager_InstanceCounter > 0 THEN
	;
ELSE
	_internal.InterfaceManager_InstanceCounter := 1;
END_IF
END_METHOD

METHOD get_terminal_id : BOOL
VAR_INPUT
	terminal_name: STRING;
END_VAR
VAR_OUTPUT
	terminal_id : uint;
	errId: HAL_ErrorEnum;
END_VAR
VAR
	i: UINT;
END_VAR
FOR i:=1 TO NUMBER_OF_TERMINALS DO
	IF terminals[i] = terminal_name THEN
		terminal_id := i;
		get_terminal_id := TRUE;
		RETURN;
	END_IF
END_FOR
get_terminal_id := FALSE;
errId := HAL_ErrorEnum.terminal_not_found;
END_METHOD

METHOD register_I_AI_Percentage : BOOL
VAR_INPUT
	interface_to_be_registered		: I_AI_Percentage;
	terminal_id 					: UINT;
	channel_number 					: USINT; 
END_VAR
VAR
	i: UINT;
END_VAR
VAR_OUTPUT
	errId		: HAL_ErrorEnum;
END_VAR
register_I_AI_Percentage:=FALSE;
IF registrations_in_cycle >= MAX_REGISTRATIONS_PER_CYCLE THEN
	register_I_AI_Percentage := FALSE;
	errId := HAL_ErrorEnum.max_registration_limit_per_cycle_reached;
	RETURN;
ELSE
	registrations_in_cycle := registrations_in_cycle + 1; 
END_IF

IF interface_to_be_registered = 0 THEN
	errId := HAL_ErrorEnum.interface_can_not_be_null;
ELSIF terminal_id = 0 THEN
	errId := HAL_ErrorEnum.terminal_name_can_not_be_empty;
ELSIF channel_number = 0 THEN
	errId := HAL_ErrorEnum.channel_number_out_of_range;
ELSE
	FOR i:=0 TO NUMBER_OF_I_AI_Percentage_INTERFACES DO
		IF I_AI_Percentage_interfaces[i].registered_interface = 0 THEN
			I_AI_Percentage_interfaces[i].channel_number 		:= channel_number;
			I_AI_Percentage_interfaces[i].registered_interface 	:= interface_to_be_registered;
			I_AI_Percentage_interfaces[i].terminal_id 			:= terminal_id;
			register_I_AI_Percentage:=TRUE;
			RETURN;
		END_IF
	END_FOR
	errId := HAL_ErrorEnum.no_empty_space_found_in_register;
END_IF
END_METHOD

METHOD register_I_AI_Temperature : BOOL
VAR_INPUT
	interface_to_be_registered      : I_AI_Temperature;
	terminal_id                     : UINT;
	channel_number                  : USINT; 
END_VAR
VAR
	i: UINT;
END_VAR
VAR_OUTPUT
	errId		: HAL_ErrorEnum;
END_VAR
END_METHOD

METHOD register_I_AI_Voltage : BOOL
VAR_INPUT
	interface_to_be_registered      : I_AI_Voltage;
	terminal_id                     : UINT;
	channel_number                  : USINT; 
END_VAR
VAR
	i: UINT;
END_VAR
VAR_OUTPUT
	errId		: HAL_ErrorEnum;
END_VAR
register_I_AI_Voltage:=FALSE;
IF registrations_in_cycle >= MAX_REGISTRATIONS_PER_CYCLE THEN
	register_I_AI_Voltage := FALSE;
	errId := HAL_ErrorEnum.max_registration_limit_per_cycle_reached;
	RETURN;
ELSE
	registrations_in_cycle := registrations_in_cycle + 1; 
END_IF

IF interface_to_be_registered = 0 THEN
	errId := HAL_ErrorEnum.interface_can_not_be_null;
ELSIF terminal_id = 0 THEN
	errId := HAL_ErrorEnum.terminal_name_can_not_be_empty;
ELSIF channel_number = 0 THEN
	errId := HAL_ErrorEnum.channel_number_out_of_range;
ELSE
	FOR i:=0 TO NUMBER_OF_I_HAL_AI_Voltage_INTERFACES DO
		IF I_AI_Voltage_interfaces[i].registered_interface = 0 THEN
			I_AI_Voltage_interfaces[i].channel_number 		:= channel_number;
			I_AI_Voltage_interfaces[i].registered_interface := interface_to_be_registered;
			I_AI_Voltage_interfaces[i].terminal_id 			:= terminal_id;
			register_I_AI_Voltage:=TRUE;
			RETURN;
		END_IF
	END_FOR
	errId := HAL_ErrorEnum.no_empty_space_found_in_register;
END_IF
END_METHOD

METHOD register_I_AO_Percentage : BOOL
VAR_INPUT
	interface_to_be_registered	: I_AO_Percentage;
	terminal_id	: UINT;
	channel_number	: USINT;
END_VAR
VAR_OUTPUT
	errId	: HAL_ErrorEnum;
END_VAR
END_METHOD

METHOD register_I_AO_Voltage : BOOL
VAR_INPUT
	interface_to_be_registered	: I_AO_Voltage;
	terminal_id	: UINT;
	channel_number	: USINT;
END_VAR
VAR_OUTPUT
	errId	: HAL_ErrorEnum;
END_VAR
VAR
	i: UINT;
END_VAR
register_I_AO_Voltage:=FALSE;
IF registrations_in_cycle >= MAX_REGISTRATIONS_PER_CYCLE THEN
	register_I_AO_Voltage := FALSE;
	errId := HAL_ErrorEnum.max_registration_limit_per_cycle_reached;
	RETURN;
ELSE
	registrations_in_cycle := registrations_in_cycle + 1; 
END_IF

IF interface_to_be_registered = 0 THEN
	errId := HAL_ErrorEnum.interface_can_not_be_null;
ELSIF terminal_id = 0 THEN
	errId := HAL_ErrorEnum.terminal_name_can_not_be_empty;
ELSIF channel_number = 0 THEN
	errId := HAL_ErrorEnum.channel_number_out_of_range;
ELSE
	FOR i:=0 TO NUMBER_OF_I_AI_Percentage_INTERFACES DO
		IF I_AO_Voltage_interfaces[i].registered_interface = 0 THEN
			I_AO_Voltage_interfaces[i].channel_number 		:= channel_number;
			I_AO_Voltage_interfaces[i].registered_interface := interface_to_be_registered;
			I_AO_Voltage_interfaces[i].terminal_id 			:= terminal_id;
			register_I_AO_Voltage:=TRUE;
			RETURN;
		END_IF
	END_FOR
	errId := HAL_ErrorEnum.no_empty_space_found_in_register;
END_IF
END_METHOD

METHOD register_terminal : BOOL
VAR_INPUT
	terminal_name : STRING;
END_VAR
VAR_OUTPUT
	errId : HAL_ErrorEnum;
    terminalId : UINT;
END_VAR
VAR
	i: UINT;
END_VAR
FOR i:=1 TO NUMBER_OF_TERMINALS DO
	IF len(terminals[i]) = 0 THEN
		terminals[i] := terminal_name;
        terminalId := i;
		register_terminal := TRUE;
		RETURN;
	END_IF
	errId := HAL_ErrorEnum.no_empty_space_found_in_register;
END_FOR
register_terminal:=FALSE;
END_METHOD

METHOD release_I_AI_Percentage : BOOL
VAR_INPUT
END_VAR
END_METHOD

METHOD request_I_AI_Percentage : BOOL
VAR_INPUT
	terminal_id                 : UINT;
	channel_number              : USINT; 
	device_id                   : UINT;
END_VAR
VAR_OUTPUT
	_interface	: I_AI_Percentage;
	errId	    : HAL_ErrorEnum;
END_VAR
VAR
	i :UINT;
END_VAR
request_I_AI_Percentage:=FALSE;

IF channel_number = 0 THEN
	errId := HAL_ErrorEnum.channel_number_out_of_range;
ELSIF device_id = 0 THEN
	errId := HAL_ErrorEnum.device_id_can_not_be_null;
ELSE

	FOR i:=0 TO NUMBER_OF_I_AI_Percentage_INTERFACES DO
		IF  I_AI_Percentage_interfaces[i].registered_interface <> 0 AND
			I_AI_Percentage_interfaces[i].terminal_id = terminal_id AND
			I_AI_Percentage_interfaces[i].channel_number = channel_number  
		THEN
			IF I_AI_Percentage_interfaces[i].connected_device_id = 0 THEN
				I_AI_Percentage_interfaces[i].connected_device_id 	:= device_id;
				_interface := I_AI_Percentage_interfaces[i].registered_interface;
				request_I_AI_Percentage:=TRUE;
			ELSE		
				errId := HAL_ErrorEnum.interface_already_in_use;
			END_IF
			RETURN;
		END_IF
	END_FOR
	errId := HAL_ErrorEnum.requested_interface_not_found;
END_IF
END_METHOD

METHOD request_I_AI_Voltage : BOOL
VAR_INPUT
	terminal_name 					: STRING;
	channel_number 					: USINT; 
	device_id						: UINT;
END_VAR
VAR_OUTPUT
	_interface	: I_AI_Voltage;
	errId	    : HAL_ErrorEnum;
END_VAR
VAR
	i :UINT;
	terminal_id: UINT;
END_VAR
IF terminal_name = '' THEN
	errId := HAL_ErrorEnum.terminal_name_can_not_be_empty;
ELSIF channel_number = 0 THEN
	errId := HAL_ErrorEnum.channel_number_out_of_range;
ELSIF device_id = 0 THEN
	errId := HAL_ErrorEnum.device_id_can_not_be_null;
ELSE
	THIS^.get_terminal_id(terminal_name, terminal_id=>terminal_id, errId=>errId);
	IF errId <> 0 THEN
		RETURN; 
	END_IF
	FOR i:=0 TO NUMBER_OF_I_HAL_AI_Voltage_INTERFACES DO
		IF  I_AI_Voltage_interfaces[i].registered_interface <> 0 AND
			I_AI_Voltage_interfaces[i].terminal_id = terminal_id AND
			I_AI_Voltage_interfaces[i].channel_number = channel_number  
		THEN
			IF I_AI_Percentage_interfaces[i].connected_device_id = 0 THEN
				errId := HAL_ErrorEnum.interface_already_in_use;
			ELSE		
				I_AI_Percentage_interfaces[i].connected_device_id 	:= device_id;
				_interface := I_AI_Voltage_interfaces[i].registered_interface;
			END_IF
			EXIT;
		END_IF
	END_FOR
	errId := HAL_ErrorEnum.requested_interface_not_found;
END_IF
END_METHOD

END_FUNCTION_BLOCK

// ---- _internal/CoE/CoE_communication_handler.TcPOU
(**
This function bock handles ADS read and write requests.
To read or write an ADS property pass an object that implements the "I_CoE_property" interface through the "add_read_request" or "add_write_request" method.
All requests will be added to an internal read or write buffer and executed one by one.
The object will be updated through the callback interface when the read or write process is done.
*)
FUNCTION_BLOCK CoE_communication_handler IMPLEMENTS I_CoE_communication_handler
VAR_INPUT
	amsNetId	: T_AmsNetId;
END_VAR
VAR_OUTPUT
END_VAR
VAR
	// ==  read  ================================== 
	done_reading_coe		: f_trig;
	CoE_property_to_read	: I_CoE_property;
	read_requests_table 	: ring_buffer_CoE_read; 
	
	coe_read 	: FB_EcCoESdoRead;	
	
	_readState		: INT;
	_executeRead	: BOOL;
	_readBuffer		: CoE_buffer_type_cast_union;
	
	// ==  write  ================================== 
	done_writing_coe		: f_trig;
	CoE_property_to_write	: I_CoE_property;
	write_requests_table 	: ring_buffer_CoE_read; 
	
	coe_write 	: FB_EcCoESdoWrite;	
	
	_writeState			: INT;
	_executeWrite		: BOOL;
	_writeBuffer		: CoE_buffer_type_cast_union;

END_VAR

// ===========================
// handle read requests
// ===
CASE _readState OF 
	0:
		IF read_requests_table.read(data=> CoE_property_to_read)THEN 
			_executeRead := TRUE;
			_readState := 10;			
		END_IF

	10:
		IF done_reading_coe.q THEN
			CoE_property_to_read.handle_read_callback(pt_buffer:=ADR(_readBuffer), errId:=coe_read.nErrId);
			_executeRead:=FALSE;
			_readState := 0;
		END_IF
ELSE
	_readState := 0;
END_CASE

IF CoE_property_to_read <> 0 THEN
	coe_read(
		sNetId		:= amsNetId, 
		nSlaveAddr	:= CoE_property_to_read.SlaveAddress, 
		nSubIndex	:= CoE_property_to_read.SubIndex, 
		nIndex		:= CoE_property_to_read.Index, 
		pDstBuf		:= ADR(_readBuffer._values), 
		cbBufLen	:= SIZEOF(_readBuffer._values), 
		bExecute	:= _executeRead, 
		tTimeout	:= , 
		bBusy		=> , 
		bError		=> , 
		nErrId		=> , 
		cbRead		=> );
		
	done_reading_coe(clk:=coe_read.bBusy);
END_IF


// ===========================
// hadndle write requests
// ===
CASE _writeState OF 
	0:
		IF write_requests_table.read(data=> CoE_property_to_write) THEN 
			_writeBuffer := CoE_property_to_write.valueToWrite;
			_executeWrite := TRUE;
			_writeState := 10;			
		END_IF

	10:
		IF done_writing_coe.q THEN
			CoE_property_to_write.handle_write_callback(errId:=coe_write.nErrId);
			_executeWrite:=FALSE;
			_writeState := 0;
		END_IF
ELSE
	_readState := 0;
END_CASE

IF CoE_property_to_write <> 0 THEN
	coe_write(
		sNetId		:= amsNetId, 
		nSlaveAddr	:= CoE_property_to_write.SlaveAddress, 
		nSubIndex	:= CoE_property_to_write.SubIndex, 
		nIndex		:= CoE_property_to_write.Index, 
		pSrcBuf		:= ADR(_writeBuffer._values), 
		cbBufLen	:= CoE_property_to_write.dataTypeSize, 
		bExecute	:= _executeWrite, 
		tTimeout	:= , 
		bBusy		=> , 
		bError		=> , 
		nErrId		=> );
		
	done_writing_coe(clk:=coe_write.bBusy);
END_IF
// ===========================

METHOD add_read_request : BOOL
VAR_INPUT
	request	: I_CoE_property;
END_VAR

IF request <> 0 THEN
	add_read_request:= THIS^.read_requests_table.write(request);
ELSE
	add_read_request:=FALSE;
END_IF
END_METHOD

METHOD add_write_request : BOOL
VAR_INPUT
	request	: I_CoE_property;
END_VAR

IF request <> 0 THEN
	add_write_request:= THIS^.write_requests_table.write(request);
ELSE
	add_write_request:=FALSE;
END_IF
END_METHOD

END_FUNCTION_BLOCK

// ---- _internal/CoE/buffer/ring_buffer_CoE_read.TcPOU
FUNCTION_BLOCK ring_buffer_CoE_read
VAR_INPUT
END_VAR
VAR_OUTPUT
END_VAR
VAR
    buffer : ARRAY[0..BUFFER_UPPER_BOUND] OF I_CoE_property;
    
    write_index: UDINT;
    read_index: UDINT;

	is_full_flag: BOOL;
END_VAR
VAR_IN_OUT
	// buffer : ARRAY[*] OF LWORD;
END_VAR
VAR CONSTANT 
    BUFFER_UPPER_BOUND : UINT:=50;
	BUFFER_CAPACITY : UINT:=BUFFER_UPPER_BOUND + 1;
END_VAR

PROPERTY capacity : uint
GET
capacity:= THIS^.buffer_capacity;
END_GET
END_PROPERTY

METHOD clear : BOOL
VAR
	i: UINT;
END_VAR

FOR i:=0 TO BUFFER_UPPER_BOUND DO
	buffer[i] :=0;  
END_FOR

write_index:=0;
read_index:=0;
is_full_flag:=FALSE;
clear:=TRUE;
END_METHOD

METHOD is_empty : BOOL
is_empty:= write_index = read_index AND NOT is_full_flag;
END_METHOD

METHOD is_full : BOOL
VAR_INPUT
END_VAR
is_full:= is_full_flag;
END_METHOD

PROPERTY level : uint
GET
VAR
	tmp: INT;
END_VAR

tmp := UDINT_TO_INT(write_index) - UDINT_TO_INT(read_index);

IF tmp < 0 THEN
    level := INT_TO_UINT(tmp + UINT_TO_INT(buffer_capacity));
ELSIF tmp = 0 AND is_full_flag THEN
    level := buffer_capacity;
ELSE
    level := INT_TO_UINT(tmp);
END_IF
END_GET
END_PROPERTY

METHOD read : BOOL
VAR_OUTPUT
	data	: I_CoE_property;
END_VAR
IF NOT THIS^.is_empty() THEN
	data:= buffer[read_index];

    read_index:= (read_index + 1) MOD buffer_capacity;
    is_full_flag:=FALSE;
    read:=TRUE;
ELSE
    read:= FALSE;
END_IF
END_METHOD

METHOD write : BOOL
VAR_INPUT
	data	: I_CoE_property;
END_VAR
IF NOT THIS^.is_full() THEN
    buffer[write_index]:= data;
    write_index:= (write_index + 1) MOD buffer_capacity;
    is_full_flag:= write_index = read_index;
    write:=TRUE;
ELSE
    write:= FALSE;
END_IF
END_METHOD

END_FUNCTION_BLOCK

// ---- digital_input/EL1808.TcPOU
(**
This function block abstracts the Beckhoff EtherCAT terminal EL1808
*)
FUNCTION_BLOCK EL1808 IMPLEMENTS I_terminal_execution
VAR_INPUT
END_VAR
VAR_OUTPUT
	DI_channel_1 		: I_HAL_DI :=_channel_1;
	DI_channel_2 		: I_HAL_DI :=_channel_2;
	DI_channel_3 		: I_HAL_DI :=_channel_3;
	DI_channel_4 		: I_HAL_DI :=_channel_4;
	DI_channel_5 		: I_HAL_DI :=_channel_5;
	DI_channel_6 		: I_HAL_DI :=_channel_6;
	DI_channel_7 		: I_HAL_DI :=_channel_7;
	DI_channel_8 		: I_HAL_DI :=_channel_8;
END_VAR
VAR
	WcState_WcState			AT%I*: BOOL;
	WcState_InputToggle		AT%I*: BOOL;
	InfoData_State			AT%I*: UINT;
	
	Channel_1_Input         AT%I*: BOOL;
	Channel_2_Input         AT%I*: BOOL;
	Channel_3_Input         AT%I*: BOOL;
	Channel_4_Input         AT%I*: BOOL;
	Channel_5_Input         AT%I*: BOOL;
	Channel_6_Input         AT%I*: BOOL;
	Channel_7_Input         AT%I*: BOOL;
	Channel_8_Input         AT%I*: BOOL;
	
	_channel_1 : HAL_DI_Channel(channel_number:=1);
	_channel_2 : HAL_DI_Channel(channel_number:=2);
	_channel_3 : HAL_DI_Channel(channel_number:=3);
	_channel_4 : HAL_DI_Channel(channel_number:=4);
	_channel_5 : HAL_DI_Channel(channel_number:=5);
	_channel_6 : HAL_DI_Channel(channel_number:=6);
	_channel_7 : HAL_DI_Channel(channel_number:=7);
	_channel_8 : HAL_DI_Channel(channel_number:=8);
END_VAR
VAR CONSTANT	
    HARDWARE_REVSION : UINT:=19;
END_VAR


_channel_1.wcState:= NOT  WcState_WcState;
_channel_2.wcState:= NOT  WcState_WcState;
_channel_3.wcState:= NOT  WcState_WcState;
_channel_4.wcState:= NOT  WcState_WcState;
_channel_5.wcState:= NOT  WcState_WcState;
_channel_6.wcState:= NOT  WcState_WcState;
_channel_7.wcState:= NOT  WcState_WcState;
_channel_8.wcState:= NOT  WcState_WcState;

_channel_1();
_channel_2();
_channel_3();
_channel_4();
_channel_5();
_channel_6();
_channel_7();
_channel_8();

_channel_1.terminal_value:=Channel_1_Input;
_channel_2.terminal_value:=Channel_2_Input;
_channel_3.terminal_value:=Channel_3_Input;
_channel_4.terminal_value:=Channel_4_Input;
_channel_5.terminal_value:=Channel_5_Input;
_channel_6.terminal_value:=Channel_6_Input;
_channel_7.terminal_value:=Channel_7_Input;
_channel_8.terminal_value:=Channel_8_Input;

METHOD FB_init : BOOL
VAR_INPUT
	bInitRetains : BOOL; // if TRUE, the retain variables are initialized (warm start / cold start)
	bInCopyCode : BOOL;  // if TRUE, the instance afterwards gets moved into the copy code (online change)
	CoE_communication_handler: I_CoE_communication_handler;
END_VAR
END_METHOD

METHOD run : BOOL
VAR_INPUT
END_VAR
THIS^();
END_METHOD

END_FUNCTION_BLOCK

// ---- digital_input/_internal/HAL_DI_Channel.TcPOU
FUNCTION_BLOCK HAL_DI_Channel IMPLEMENTS I_HAL_DI
VAR_INPUT
	terminal_address		: WORD;
END_VAR
VAR_OUTPUT
END_VAR
VAR
	_errId:UINT;
	_xValue: BOOL;
	_channel_number: UINT;
END_VAR

PROPERTY errId : UINT
GET
errId := _errId;
END_GET
END_PROPERTY

METHOD FB_init : BOOL
VAR_INPUT
	bInitRetains 	: BOOL; // if TRUE, the retain variables are initialized (warm start / cold start)
	bInCopyCode 	: BOOL;  // if TRUE, the instance afterwards gets moved into the copy code (online change)
    channel_number  : UINT;
END_VAR

_channel_number :=channel_number;
END_METHOD

PROPERTY terminal_value : bool
SET
_xValue:=terminal_value;
END_SET
END_PROPERTY

PROPERTY WcState : bool
GET
END_GET
SET
END_SET
END_PROPERTY

PROPERTY xValue : BOOL
GET
xValue:=_xValue;
END_GET
END_PROPERTY

END_FUNCTION_BLOCK

// ---- digital_output/EL2808.TcPOU
(**
This function block abstracts the Beckhoff EtherCAT terminal EL2808
*)
FUNCTION_BLOCK EL2808 IMPLEMENTS I_terminal_execution
VAR_INPUT
END_VAR
VAR_OUTPUT
	DO_channel_1 		: I_HAL_DO :=_channel_1;
	DO_channel_2 		: I_HAL_DO :=_channel_2;
	DO_channel_3 		: I_HAL_DO :=_channel_3;
	DO_channel_4 		: I_HAL_DO :=_channel_4;
	DO_channel_5 		: I_HAL_DO :=_channel_5;
	DO_channel_6 		: I_HAL_DO :=_channel_6;
	DO_channel_7 		: I_HAL_DO :=_channel_7;
	DO_channel_8 		: I_HAL_DO :=_channel_8;
END_VAR
VAR
	WcState_WcState			AT%I*: BOOL;
	InfoData_State			AT%I*: UINT;
	
	Channel_1_Output         AT%Q*: BOOL;
	Channel_2_Output         AT%Q*: BOOL;
	Channel_3_Output         AT%Q*: BOOL;
	Channel_4_Output         AT%Q*: BOOL;
	Channel_5_Output         AT%Q*: BOOL;
	Channel_6_Output         AT%Q*: BOOL;
	Channel_7_Output         AT%Q*: BOOL;
	Channel_8_Output         AT%Q*: BOOL;
	
	_channel_1 : HAL_DO_Channel(channel_number:=1);
	_channel_2 : HAL_DO_Channel(channel_number:=2);
	_channel_3 : HAL_DO_Channel(channel_number:=3);
	_channel_4 : HAL_DO_Channel(channel_number:=4);
	_channel_5 : HAL_DO_Channel(channel_number:=5);
	_channel_6 : HAL_DO_Channel(channel_number:=6);
	_channel_7 : HAL_DO_Channel(channel_number:=7);
	_channel_8 : HAL_DO_Channel(channel_number:=8);
END_VAR
VAR CONSTANT	
    HARDWARE_REVSION : UINT:=19;
END_VAR


_channel_1.wcState:= NOT  WcState_WcState;
_channel_2.wcState:= NOT  WcState_WcState;
_channel_3.wcState:= NOT  WcState_WcState;
_channel_4.wcState:= NOT  WcState_WcState;
_channel_5.wcState:= NOT  WcState_WcState;
_channel_6.wcState:= NOT  WcState_WcState;
_channel_7.wcState:= NOT  WcState_WcState;
_channel_8.wcState:= NOT  WcState_WcState;

_channel_1();
_channel_2();
_channel_3();
_channel_4();
_channel_5();
_channel_6();
_channel_7();
_channel_8();

Channel_1_Output := _channel_1.terminal_value;
Channel_2_Output := _channel_2.terminal_value;
Channel_3_Output := _channel_3.terminal_value;
Channel_4_Output := _channel_4.terminal_value;
Channel_5_Output := _channel_5.terminal_value;
Channel_6_Output := _channel_6.terminal_value;
Channel_7_Output := _channel_7.terminal_value;
Channel_8_Output := _channel_8.terminal_value;

METHOD FB_init : BOOL
VAR_INPUT
	bInitRetains : BOOL; // if TRUE, the retain variables are initialized (warm start / cold start)
	bInCopyCode : BOOL;  // if TRUE, the instance afterwards gets moved into the copy code (online change)
	CoE_communication_handler : I_CoE_communication_handler;
END_VAR
END_METHOD

METHOD run : BOOL
VAR_INPUT
END_VAR
THIS^();
END_METHOD

END_FUNCTION_BLOCK

// ---- digital_output/_internal/HAL_DO_Channel.TcPOU
FUNCTION_BLOCK HAL_DO_Channel IMPLEMENTS I_HAL_DO
VAR_INPUT
	terminal_address		: WORD;
END_VAR
VAR_OUTPUT
END_VAR
VAR
	_terminal_value: BOOL;
	_errId:HAL_ErrorEnum;
	_xValue: BOOL;
	_channel_number: UINT;
END_VAR

PROPERTY errId : HAL_ErrorEnum
GET
errId := _errId;
END_GET
END_PROPERTY

METHOD FB_init : BOOL
VAR_INPUT
	bInitRetains 	: BOOL; // if TRUE, the retain variables are initialized (warm start / cold start)
	bInCopyCode 	: BOOL;  // if TRUE, the instance afterwards gets moved into the copy code (online change)
    channel_number  : UINT;
END_VAR

_channel_number :=channel_number;
END_METHOD

PROPERTY terminal_value : bool
GET
terminal_value := _xValue;
END_GET
END_PROPERTY

PROPERTY WcState : bool
GET
END_GET
SET
END_SET
END_PROPERTY

PROPERTY xValue : BOOL
GET
xValue:=_xValue;
END_GET
SET
_xValue := xValue;
END_SET
END_PROPERTY

END_FUNCTION_BLOCK

// ---- analog_output/voltage/EL4002.TcPOU
(**
This function block abstracts the Beckhoff EtherCAT terminal EL4002 (0…10 V, 12 Bit)
*)
FUNCTION_BLOCK EL4002 IMPLEMENTS I_terminal_execution
VAR_INPUT
END_VAR
VAR_OUTPUT
	AO_Voltage_channel_1 		: I_AO_Voltage :=_ar_channels[1];
	AO_Voltage_channel_2 		: I_AO_Voltage :=_ar_channels[2];
END_VAR
VAR
	WcState_WcState			AT%I*: BOOL;
	InfoData_State			AT%I*: UINT;
	InfoData_AdsAddr_netId  AT%I*: AMSNETID;
	InfoData_AdsAddr_port 	AT%I*: WORD;
	
	AO_Outputs_Channel_1_Analog_output         AT%Q*: INT;
	AO_Outputs_Channel_2_Analog_output         AT%Q*: INT;
	
    _ar_channels : ARRAY[1..NUMBER_OF_CHANNELS] OF AO_Voltage_Channel[
		(adc_min:=ADC_MIN, adc_max:=ADC_MAX, physical_min:=PHYSICAL_MIN, physical_max:=PHYSICAL_MAX, channel_number:=1),
		(adc_min:=ADC_MIN, adc_max:=ADC_MAX, physical_min:=PHYSICAL_MIN, physical_max:=PHYSICAL_MAX, channel_number:=2)
    ];

	// ===============================================================================
	// CoE handling  
	// ==============
    _I_CoE_com_handler      : I_CoE_communication_handler;
    _CoE_prop_handler       : CoE_property_handler;
    // ====  CoE properties  ===========
	_p_DeviceName 			: CoE_property_string(Index:=16#1008 , SubIndex:=0, writable:=FALSE, propertyType:=0, pollingInterval:=T#5S);
	_p_DeviceType 			: CoE_property_udint(Index:=16#1000 , SubIndex:=0, writable:=FALSE, propertyType:=0, pollingInterval:=T#5S);
	_p_ProductCode 			: CoE_property_udint(Index:=16#1018 , SubIndex:=2, writable:=FALSE, propertyType:=0, pollingInterval:=T#5S);
	_p_Revision 			: CoE_property_udint(Index:=16#1018 , SubIndex:=3, writable:=FALSE, propertyType:=0, pollingInterval:=T#5S);
	_p_SerialNumber 		: CoE_property_udint(Index:=16#1018 , SubIndex:=4, writable:=FALSE, propertyType:=0, pollingInterval:=T#5S);
	_p_SoftwareVersion		: CoE_property_string(Index:=16#100A , SubIndex:=0, writable:=FALSE, propertyType:=0, pollingInterval:=T#5S);
	_p_VendorId 			: CoE_property_udint(Index:=16#1018 , SubIndex:=1, writable:=FALSE, propertyType:=0, pollingInterval:=T#5S);
	_p_HardwareVersion		: CoE_property_string(Index:=16#1009 , SubIndex:=0, writable:=FALSE, propertyType:=0, pollingInterval:=T#5S);
	// ==============
	_properties  : ARRAY[1..8]OF I_CoE_property:=[
		_p_DeviceName, _p_DeviceType, _p_ProductCode, _p_Revision, _p_SerialNumber, 
		_p_SoftwareVersion, _p_VendorId, _p_HardwareVersion
	];
	// ===============================================================================
    
	_I_InterfaceManager : I_InterfaceManager;
    _terminal_name      : STRING;
    _terminal_id        : UINT;
    errId               : HAL_ErrorEnum;
	neg_wcState         : f_trig;
    _j                  : USINT;
END_VAR
VAR CONSTANT
	ADC_MIN        	: INT:=0;
	ADC_MAX        	: INT:=32767;
	PHYSICAL_MIN 	: INT:=0;
	PHYSICAL_MAX 	: INT:=10;
	
    HARDWARE_REVSION : UINT:=19;
    NUMBER_OF_CHANNELS : USINT:=2;
END_VAR


_ar_channels[1].wcState:= WcState_WcState;
_ar_channels[2].wcState:= WcState_WcState;

_ar_channels[1](terminal_address:=InfoData_AdsAddr_port, CoE_communication_handler:=_I_CoE_com_handler);
_ar_channels[2](terminal_address:=InfoData_AdsAddr_port, CoE_communication_handler:=_I_CoE_com_handler);

AO_Outputs_Channel_1_Analog_output := _ar_channels[1].terminal_value;
AO_Outputs_Channel_2_Analog_output := _ar_channels[2].terminal_value;

IF  _I_InterfaceManager <> 0 AND 
    _I_CoE_com_handler <> 0
THEN
    FOR _j:=1 TO NUMBER_OF_CHANNELS DO
        // should be possible to get rid of the address input 
        _ar_channels[_j](terminal_address:=InfoData_AdsAddr_port, CoE_communication_handler:=_I_CoE_com_handler);
    END_FOR
    
    _CoE_prop_handler(terminal_address:=InfoData_AdsAddr_port, CoE_communication_handler:=_I_CoE_com_handler, CoE_properties:=_properties);

    neg_wcState(CLK:=WcState_WcState);
    IF neg_wcState.Q THEN
        ;
    END_IF
END_IF

METHOD FB_init : BOOL
VAR_INPUT
	bInitRetains : BOOL; // if TRUE, the retain variables are initialized (warm start / cold start)
	bInCopyCode : BOOL;  // if TRUE, the instance afterwards gets moved into the copy code (online change)
	CoE_communication_handler: I_CoE_communication_handler;
    InterfaceManager            : I_InterfaceManager;
	name                        : STRING;
END_VAR

_I_CoE_com_handler := CoE_communication_handler;

FOR _j:=1 TO NUMBER_OF_CHANNELS DO
    _ar_channels[_j].CoE_communication_handler := CoE_communication_handler;
END_FOR

_terminal_name := name;
_I_InterfaceManager := InterfaceManager;

// register  terminal and all channel interfaces
IF InterfaceManager <> 0 THEN
    _I_InterfaceManager.register_terminal(terminal_name:=_terminal_name , errId=>errId , terminalId=>_terminal_id);
    
    FOR _j:=1 TO NUMBER_OF_CHANNELS DO
        _ar_channels[_j].register_channel(terminalId:=_terminal_id , I_interface_manager:=_I_InterfaceManager , errId=>errId );
        IF errId <> HAL_ErrorEnum.no_error THEN
            ;  // ToDo: add logging or Error handling 
        END_IF 
    END_FOR
END_IF
END_METHOD

METHOD run : BOOL
VAR_INPUT
END_VAR
THIS^();
END_METHOD

END_FUNCTION_BLOCK

// ---- analog_output/_internal/AO_Voltage_Channel.TcPOU
FUNCTION_BLOCK AO_Voltage_Channel IMPLEMENTS I_AO_Voltage, I_AO_percentage
VAR_INPUT
	terminal_address		    : WORD;
	CoE_communication_handler	: I_CoE_communication_handler;
END_VAR
VAR_OUTPUT
END_VAR
VAR
	_adc_min        : INT;
    _adc_max        : INT;
	_physical_min 	: INT;
	_physical_max 	: INT;
	_channel_number : USINT;
	_rValue			: REAL;
	_wcState		: BOOL;
	
    _CoE_prop_handler       : CoE_property_handler;
	// ===============================================================================
	// CoE properties 
	// ==============
	index_1 						: WORD:= 16#8000 + INT_TO_WORD(_CoE_channel_offset);
	_p_Enable_user_scale    		: CoE_property_bool(Index:=index_1 , SubIndex:=1, writable:=TRUE, propertyType:=0, pollingInterval:=T#5S);
	_p_Presentation 				: CoE_property_usint(Index:=index_1 , SubIndex:=2, writable:=TRUE, propertyType:=0, pollingInterval:=T#5S);			// DT0800EN03
	_p_Watchdog 					: CoE_property_usint(Index:=index_1 , SubIndex:=5, writable:=TRUE, propertyType:=0, pollingInterval:=T#5S);			// DT0801EN02
	_p_Enable_user_calibration  	: CoE_property_bool(Index:=index_1 , SubIndex:=7, writable:=TRUE, propertyType:=0, pollingInterval:=T#5S);
	_p_Enable_vendor_calibration    : CoE_property_bool(Index:=index_1 , SubIndex:=8, writable:=TRUE, propertyType:=0, pollingInterval:=T#5S);
	_p_Offset   					: CoE_property_int(Index:=index_1 , SubIndex:=17, writable:=TRUE, propertyType:=0, pollingInterval:=T#5S);
	_p_Gain 						: CoE_property_dint(Index:=index_1 , SubIndex:=18, writable:=TRUE, propertyType:=0, pollingInterval:=T#5S);
	_p_Default_output   			: CoE_property_int(Index:=index_1 , SubIndex:=19, writable:=TRUE, propertyType:=0, pollingInterval:=T#5S);
	_p_Default_output_ramp  		: CoE_property_uint(Index:=index_1 , SubIndex:=20, writable:=TRUE, propertyType:=0, pollingInterval:=T#5S);
	_p_User_calibration_offset  	: CoE_property_int(Index:=index_1 , SubIndex:=21, writable:=TRUE, propertyType:=0, pollingInterval:=T#5S);
	_p_User_calibration_gain    	: CoE_property_uint(Index:=index_1 , SubIndex:=22, writable:=TRUE, propertyType:=0, pollingInterval:=T#5S);
	// ==============
	_properties  : ARRAY[1..11]OF I_CoE_property:=[
		_p_Enable_user_scale, _p_Presentation, _p_Watchdog, _p_Enable_user_calibration, _p_Enable_vendor_calibration, _p_Offset,
		_p_Gain, _p_Default_output, _p_Default_output_ramp, _p_User_calibration_offset, _p_User_calibration_gain];
	// ===============================================================================
	_CoE_channel_offset: INT;
	i: UINT;
	_init_done: BOOL;
	_init_step: INT:=1;
	_old_init_step: INT;

	_errId: HAL_ErrorEnum;

	//  ====  I_AI_percentage  ====
	_max_value 	: REAL:=10.0;
	_min_value 	: REAL:=0.0;
	_value      : REAL;
END_VAR

// CoE Property handling 
_CoE_prop_handler(terminal_address:=terminal_address, CoE_communication_handler:=CoE_communication_handler, CoE_properties:=_properties);

// =========================================
(*
IF NOT _wcState THEN 
	_init_step:=1;
	_old_init_step:=0;
	_init_done:=FALSE;
	FOR i:=1 TO MAX_NUMBER_OF_PROPERTIES DO
		IF _properties[i] <> 0 THEN
			_properties[i].reinit();
		ELSE
			EXIT;
		END_IF
	END_FOR
END_IF
*)

PROPERTY errId : HAL_ErrorEnum
GET
errId := _errId;
END_GET
END_PROPERTY

METHOD FB_init : BOOL
VAR_INPUT
	bInitRetains 	: BOOL; // if TRUE, the retain variables are initialized (warm start / cold start)
	bInCopyCode 	: BOOL;  // if TRUE, the instance afterwards gets moved into the copy code (online change)
    adc_min         : INT;
    adc_max         : INT;
	physical_min 	: INT;
	physical_max 	: INT;
	channel_number  : USINT;
END_VAR

VAR
	i: UINT;
END_VAR

_adc_min        := adc_min;
_adc_max        := adc_max;
_physical_min 	:= physical_min;
_physical_max 	:= physical_max;
_channel_number :=channel_number;

CASE channel_number OF
	1:
		_CoE_channel_offset:=16#0;
	2:
		_CoE_channel_offset:=16#10;
	3:
		_CoE_channel_offset:=16#20;
	4:
		_CoE_channel_offset:=16#30;
END_CASE
END_METHOD

METHOD get_Default_output : BOOL
VAR_OUTPUT
	value	: INT;
END_VAR
get_Default_output:=_p_Default_output.get_value(value=>value, errId => );
END_METHOD

METHOD get_Default_output_ramp : BOOL
VAR_OUTPUT
	value	: UINT;
END_VAR
get_Default_output_ramp:=_p_Default_output_ramp.get_value(value=>value, errId => );
END_METHOD

METHOD get_Enable_user_calibration : BOOL
VAR_OUTPUT
	value	: BOOL;
END_VAR
get_Enable_user_calibration:=_p_Enable_user_calibration.get_value(value=>value, errId => );
END_METHOD

METHOD get_Enable_user_scale : BOOL
VAR_OUTPUT
	value	: BOOL;
END_VAR
get_Enable_user_scale:=_p_Enable_user_scale.get_value(value=>value, errId => );
END_METHOD

METHOD get_Enable_vendor_calibration : BOOL
VAR_OUTPUT
	value	: BOOL;
END_VAR
get_Enable_vendor_calibration:=_p_Enable_vendor_calibration.get_value(value=>value, errId => );
END_METHOD

METHOD get_Gain : BOOL
VAR_OUTPUT
	value	: DINT;
END_VAR
get_Gain:=_p_Gain.get_value(value=>value, errId => );
END_METHOD

METHOD get_Offset : BOOL
VAR_OUTPUT
	value	: INT;
END_VAR
get_Offset:=_p_Offset.get_value(value=>value, errId => );
END_METHOD

METHOD get_Presentation : BOOL
VAR_OUTPUT
	value	: ENU_DT0801EN03;
END_VAR

VAR
	tmp: USINT;
END_VAR
get_Presentation:=_p_Presentation.get_value(value=>tmp, errId => );
value:=USINT_TO_INT(tmp);
END_METHOD

METHOD get_User_calibration_gain : BOOL
VAR_OUTPUT
	value	: UINT;
END_VAR
get_User_calibration_gain:=_p_User_calibration_gain.get_value(value=>value, errId => );
END_METHOD

METHOD get_User_calibration_offset : BOOL
VAR_OUTPUT
	value	: INT;
END_VAR
get_User_calibration_offset:=_p_User_calibration_offset.get_value(value=>value, errId => );
END_METHOD

METHOD get_Watchdog : BOOL
VAR_OUTPUT
	value	: ENU_DT0800EN02;
END_VAR

VAR
	tmp: USINT;
END_VAR
get_Watchdog:=_p_Watchdog.get_value(value=>tmp, errId => );
value := USINT_TO_INT(tmp);
END_METHOD

PROPERTY max_value : REAL
GET
max_value := _max_value;
END_GET
SET
IF max_value <= 0 THEN
	_max_value := 0.0001;
ELSE
	_max_value := max_value;
END_IF
END_SET
END_PROPERTY

PROPERTY min_value : REAL
GET
min_value := _min_value;
END_GET
SET
_min_value := min_value;
END_SET
END_PROPERTY

METHOD register_channel : BOOL
VAR_INPUT
    terminalId : UINT;
    I_interface_manager : I_interfaceManager;
END_VAR
VAR_OUTPUT
	errId		: HAL_ErrorEnum;
END_VAR
THIS^.register_I_AO_percentage(terminalId:=terminalId , I_interface_manager:=I_interface_manager , errId=>errId );
IF errId = HAL_ErrorEnum.no_error THEN
	THIS^.register_I_AO_Voltage(terminalId:=terminalId , I_interface_manager:=I_interface_manager , errId=>errId );
END_IF
END_METHOD

METHOD register_I_AO_percentage : BOOL
VAR_INPUT
    terminalId : UINT;
    I_interface_manager : I_interfaceManager;
END_VAR
VAR_OUTPUT
	errId		: HAL_ErrorEnum;
END_VAR
register_I_AO_percentage:= I_interface_manager.register_I_AO_Percentage(THIS^, terminalId, channel_number := THIS^._channel_number, errId=>errId);
END_METHOD

METHOD register_I_AO_Voltage : BOOL
VAR_INPUT
    terminalId : UINT;
    I_interface_manager : I_interfaceManager;
END_VAR
VAR_OUTPUT
	errId		: HAL_ErrorEnum;
END_VAR
register_I_AO_Voltage:= I_interface_manager.register_I_AO_Voltage(THIS^, terminalId, channel_number := THIS^._channel_number, errId=>errId);
END_METHOD

PROPERTY rValue : REAL
GET
rValue:=_rValue;
END_GET
SET
IF rValue < DINT_TO_REAL(_physical_min) THEN
	_errId := 6;
ELSIF rValue > DINT_TO_REAL(_physical_max) THEN
	_errId := 7;
ELSE
	_rValue := rValue;
END_IF
END_SET
END_PROPERTY

METHOD set_Default_output : BOOL
VAR_INPUT
	value	: INT;
END_VAR
set_Default_output:=_p_Default_output.set_value(value:=value);
END_METHOD

METHOD set_Default_output_ramp : BOOL
VAR_INPUT
	value	: UINT;
END_VAR
set_Default_output_ramp:=_p_Default_output_ramp.set_value(value:=value);
END_METHOD

METHOD set_Enable_user_calibration : BOOL
VAR_INPUT
	value	: BOOL;
END_VAR
set_Enable_user_calibration:=_p_Enable_user_calibration.set_value(value:=value);
END_METHOD

METHOD set_Enable_user_scale : BOOL
VAR_INPUT
	value	: BOOL;
END_VAR
set_Enable_user_scale:=_p_Enable_user_scale.set_value(value:=value);
END_METHOD

METHOD set_Enable_vendor_calibration : BOOL
VAR_INPUT
	value	: BOOL;
END_VAR
set_Enable_vendor_calibration:=_p_Enable_vendor_calibration.set_value(value:=value);
END_METHOD

METHOD set_Gain : BOOL
VAR_INPUT
	value	: DINT;
END_VAR
set_Gain:=_p_Gain.set_value(value:=value);
END_METHOD

METHOD set_Offset : BOOL
VAR_INPUT
	value	: INT;
END_VAR
set_Offset:=_p_Offset.set_value(value:=value);
END_METHOD

METHOD set_Presentation : BOOL
VAR_INPUT
	value	: ENU_DT0801EN03;
END_VAR
set_Presentation:=_p_Presentation.set_value(value:=INT_TO_USINT(value));
END_METHOD

METHOD set_User_calibration_gain : BOOL
VAR_INPUT
	value	: UINT;
END_VAR
set_User_calibration_gain:=_p_User_calibration_gain.set_value(value:=value);
END_METHOD

METHOD set_User_calibration_offset : BOOL
VAR_INPUT
	value	: INT;
END_VAR
set_User_calibration_offset:=_p_User_calibration_offset.set_value(value:=value);
END_METHOD

METHOD set_Watchdog : BOOL
VAR_INPUT
	value	: ENU_DT0800EN02;
END_VAR
set_Watchdog:=_p_Watchdog.set_value(value:=int_TO_USINT(value));
END_METHOD

PROPERTY terminal_value : int
GET

linear_phy_to_adc(
	physical_min	:= _physical_min , 
	physical_max	:= _physical_max , 
	adc_min			:= _adc_min , 
	adc_max			:= _adc_max , 
	physical_value	:= rValue , 
	adc_value		=> terminal_value , 
	errId			=> _errId 
);
	
(*
linear_phy_to_adc(
	physical_min	:= 0 , 
	physical_max	:= 100 , 
	adc_min			:= REAL_TO_INT(_min_value) , 
	adc_max			:= REAL_TO_INT(_max_value) , 
	physical_value	:= _value , 
	adc_value		=> terminal_value , 
	errId			=> _errId 
);
*)
END_GET
END_PROPERTY

PROPERTY value : REAL
GET
value := _value;
END_GET
END_PROPERTY

PROPERTY wcState : bool
GET
wcState:=_wcState;
END_GET
SET
_wcState:=wcState;
END_SET
END_PROPERTY

END_FUNCTION_BLOCK

// ---- _internal/CoE/CoE_property_handler.TcPOU
FUNCTION_BLOCK FINAL CoE_property_handler
VAR_INPUT
    terminal_address            :  WORD;
    CoE_communication_handler   : I_CoE_communication_handler;
END_VAR
VAR_OUTPUT
END_VAR
VAR
    // _I_CoE_com_handler : I_CoE_communication_handler;
	index: DINT;
    state : INT;
    propertyInitErrorCode: UDINT;
	_init_done: BOOL;
	init_index: DINT;
	number_of_properties: DINT;
END_VAR
VAR_IN_OUT
	CoE_properties: ARRAY[*] OF I_CoE_property;
END_VAR


CASE state OF 
    0:  // pre init
        init_index := LOWER_BOUND(CoE_properties, 1);
        number_of_properties :=  UPPER_BOUND(CoE_properties, 1) - LOWER_BOUND(CoE_properties, 1);
        state := 5;
        
    5:
        IF terminal_address <> 0 AND CoE_communication_handler <> 0 THEN
            FOR index := LOWER_BOUND(CoE_properties, 1) TO UPPER_BOUND(CoE_properties, 1) DO
                CoE_properties[index].SlaveAddress := terminal_address;
                CoE_properties[index].CoE_communication_handler := CoE_communication_handler;
            END_FOR	
            state := 10;
		END_IF
        
	10: // initialize all CoE-properties 
		IF CoE_properties[init_index].reinit(errId=> propertyInitErrorCode) THEN 
			// ToDo add error handling
			IF init_index < number_of_properties THEN
				init_index := init_index + 1;
			ELSE
				state := 20;
				_init_done:=TRUE; 
			END_IF
		END_IF
	
	20: // run all CoE-properties 
        FOR index := LOWER_BOUND(CoE_properties, 1) TO UPPER_BOUND(CoE_properties, 1) DO
            CoE_properties[index].run();
        END_FOR		
END_CASE

END_FUNCTION_BLOCK

// ---- _internal/CoE/properties/CoE_property_bool.TcPOU
FUNCTION_BLOCK CoE_property_bool EXTENDS CoE_property
VAR_INPUT
END_VAR
VAR_OUTPUT
END_VAR
VAR
	_value : BOOL;
END_VAR

PROPERTY dataTypeSize : UINT
GET
dataTypeSize := SIZEOF(_value);
END_GET
END_PROPERTY

METHOD get_value : BOOL
VAR_OUTPUT
	value : bool ;
	errId : UDINT;
END_VAR
IF init_done THEN
	value := _value;
	get_value := TRUE;
ELSE
	errId := 2;
	get_value := FALSE;
END_IF
END_METHOD

METHOD handle_read_callback : BOOL
VAR_INPUT
	pt_buffer : POINTER TO CoE_buffer_type_cast_union;
	errId : UDINT;
END_VAR

_value := pt_buffer^.value_bool;
_init_done:=TRUE;
_read_errId:=errId;
END_METHOD

METHOD set_value : BOOL
VAR_INPUT
	value : bool ;
END_VAR
_valueToWrite.value_bool := value;
IF THIS^._I_CoE_communication_handler <> 0 THEN 
	THIS^._I_CoE_communication_handler.add_write_request(THIS^);
ELSE
	errId:=1;
END_IF
END_METHOD

END_FUNCTION_BLOCK

// ---- _internal/CoE/properties/CoE_property.TcPOU
FUNCTION_BLOCK ABSTRACT CoE_property IMPLEMENTS I_CoE_property
VAR_INPUT
END_VAR
VAR_OUTPUT
END_VAR
VAR
	_SubIndex 		: BYTE;
	_Index			: WORD;
	_init_done		: BOOL;
	_neg_replay		: f_trig;
	_SlaveAddress	: WORD;
	_propertyType	: UINT;
	_pollingInterval: TIME;
	_I_CoE_communication_handler: I_CoE_communication_handler;
	
	_read_errId		: UDINT;
	_write_errId	: UDINT;
	_init_state		: INT;
	
	_valueToWrite 	: CoE_buffer_type_cast_union;

	pollingTimer: ton;
	
	errId: INT;
END_VAR

CASE _propertyType OF 
	0:  // cashed 
		;
	
	1:  // polling 
		pollingTimer(IN:=NOT pollingTimer.q, PT:=_pollingInterval);
		IF pollingTimer.Q THEN
			IF THIS^._I_CoE_communication_handler <> 0 THEN 
				THIS^._I_CoE_communication_handler.add_read_request(THIS^);
			ELSE
				errId:=1;
			END_IF
		END_IF
	
	2: // on request
		IF THIS^._I_CoE_communication_handler <> 0 THEN 
			THIS^._I_CoE_communication_handler.add_read_request(THIS^);
		ELSE
			errId:=1; 
		END_IF

ELSE
	errId:=2; 
END_CASE

PROPERTY CoE_communication_handler : I_CoE_communication_handler
GET
CoE_communication_handler:=_I_CoE_communication_handler;
END_GET
SET
_I_CoE_communication_handler:=CoE_communication_handler;
END_SET
END_PROPERTY

PROPERTY dataTypeSize : UINT
GET
END_GET
END_PROPERTY

METHOD FB_init : BOOL
VAR_INPUT
	bInitRetains 			: BOOL; // if TRUE, the retain variables are initialized (warm start / cold start)
	bInCopyCode 			: BOOL;  // if TRUE, the instance afterwards gets moved into the copy code (online change)
	Index					: WORD;
	SubIndex				: BYTE;
	writable				: BOOL;
	propertyType			: UINT;
	pollingInterval 		: TIME;
END_VAR
_Index:=Index;
_SubIndex:=SubIndex;
_propertyType:=propertyType;
_pollingInterval:=pollingInterval;
END_METHOD

METHOD handle_read_callback : BOOL
VAR_INPUT
	pt_buffer : POINTER TO CoE_buffer_type_cast_union;
	errId : UDINT;
END_VAR
END_METHOD

METHOD handle_write_callback : BOOL
VAR_INPUT
	errId	: UDINT;
END_VAR
_write_errId:=errId;
END_METHOD

PROPERTY Index : word
GET
Index:=_Index;
END_GET
SET
_Index:=Index;
END_SET
END_PROPERTY

PROPERTY init_done : BOOL
GET
init_done := _init_done;
END_GET
END_PROPERTY

METHOD reinit : BOOL
VAR_OUTPUT
	errId: UDINT;
END_VAR

CASE _init_state OF 
	0:  // add read request and continue
		_init_done:=FALSE;
		reinit:=FALSE;
		IF THIS^._I_CoE_communication_handler <> 0 THEN 
			THIS^._I_CoE_communication_handler.add_read_request(THIS^);
		ELSE
			errId:=1;
		END_IF
		_init_state := 10;
		
	10: // wait for read callback
		reinit:=TRUE;
		errId:=_read_errId;
		_init_state := 0;
END_CASE
END_METHOD

METHOD run : BOOL
THIS^();
END_METHOD

PROPERTY SlaveAddress : uint
GET
SlaveAddress:=_SlaveAddress;
END_GET
SET
_SlaveAddress:=SlaveAddress;
END_SET
END_PROPERTY

PROPERTY SubIndex : BYTE
GET
SubIndex:=_SubIndex;
END_GET
SET
_SubIndex:=SubIndex;
END_SET
END_PROPERTY

PROPERTY valueToWrite : CoE_buffer_type_cast_union
GET
valueToWrite := _valueToWrite;
END_GET
END_PROPERTY

END_FUNCTION_BLOCK

// ---- _internal/CoE/properties/CoE_property_usint.TcPOU
FUNCTION_BLOCK CoE_property_usint EXTENDS CoE_property
VAR_INPUT
END_VAR
VAR_OUTPUT
END_VAR
VAR
	_value : USINT;
END_VAR

SUPER^();

PROPERTY dataTypeSize : UINT
GET
dataTypeSize := SIZEOF(_value);
END_GET
END_PROPERTY

METHOD get_value : BOOL
VAR_OUTPUT
	value : usINT ;
	errId : UDINT;
END_VAR
IF init_done THEN
	value := _value;
	get_value := TRUE;
ELSE
	errId := 2;
	get_value := FALSE;
END_IF
END_METHOD

METHOD handle_read_callback : BOOL
VAR_INPUT
	pt_buffer : POINTER TO CoE_buffer_type_cast_union;
	errId : UDINT;
END_VAR

_value := pt_buffer^.value_usint;
_init_done:=TRUE;
_read_errId:=errId;
END_METHOD

METHOD set_value : BOOL
VAR_INPUT
	value : USINT ;
END_VAR
_valueToWrite.value_usint := value;
IF THIS^._I_CoE_communication_handler <> 0 THEN 
	THIS^._I_CoE_communication_handler.add_write_request(THIS^);
ELSE
	errId:=1;
END_IF
END_METHOD

END_FUNCTION_BLOCK

// ---- _internal/CoE/properties/CoE_property_int.TcPOU
FUNCTION_BLOCK CoE_property_int EXTENDS CoE_property
VAR_INPUT
END_VAR
VAR_OUTPUT
END_VAR
VAR
	_value : INT;
END_VAR

SUPER^();

PROPERTY dataTypeSize : UINT
GET
dataTypeSize := SIZEOF(_value);
END_GET
END_PROPERTY

METHOD get_value : BOOL
VAR_OUTPUT
	value : INT ;
	errId : UDINT;
END_VAR
IF init_done THEN
	value := _value;
	get_value := TRUE;
ELSE
	errId := 2;
	get_value := FALSE;
END_IF
END_METHOD

METHOD handle_read_callback : BOOL
VAR_INPUT
	pt_buffer : POINTER TO CoE_buffer_type_cast_union;
	errId : UDINT;
END_VAR

_value := pt_buffer^.value_int;
_init_done:=TRUE;
_read_errId:=errId;
END_METHOD

METHOD set_value : BOOL
VAR_INPUT
	value : int ;
END_VAR
_valueToWrite.value_int := value;
IF THIS^._I_CoE_communication_handler <> 0 THEN 
	THIS^._I_CoE_communication_handler.add_write_request(THIS^);
ELSE
	errId:=1;
END_IF
END_METHOD

END_FUNCTION_BLOCK

// ---- _internal/CoE/properties/CoE_property_dint.TcPOU
FUNCTION_BLOCK CoE_property_dint EXTENDS CoE_property
VAR_INPUT
END_VAR
VAR_OUTPUT
END_VAR
VAR
	_value : DINT;
END_VAR

SUPER^();

PROPERTY dataTypeSize : UINT
GET
dataTypeSize := SIZEOF(_value);
END_GET
END_PROPERTY

METHOD get_value : BOOL
VAR_OUTPUT
	value : DINT ;
	errId : UDINT;
END_VAR
IF init_done THEN
	value := _value;
	get_value := TRUE;
ELSE
	errId := 2;
	get_value := FALSE;
END_IF
END_METHOD

METHOD handle_read_callback : BOOL
VAR_INPUT
	pt_buffer : POINTER TO CoE_buffer_type_cast_union;
	errId : UDINT;
END_VAR

_value := pt_buffer^.value_dint;
_init_done:=TRUE;
_read_errId:=errId;
END_METHOD

METHOD set_value : BOOL
VAR_INPUT
	value : dint ;
END_VAR
_valueToWrite.value_dint := value;
IF THIS^._I_CoE_communication_handler <> 0 THEN 
	THIS^._I_CoE_communication_handler.add_write_request(THIS^);
ELSE
	errId:=1;
END_IF
END_METHOD

END_FUNCTION_BLOCK

// ---- _internal/CoE/properties/CoE_property_uint.TcPOU
FUNCTION_BLOCK CoE_property_uint EXTENDS CoE_property
VAR_INPUT
END_VAR
VAR_OUTPUT
END_VAR
VAR
	_value : UINT;
END_VAR

SUPER^();

PROPERTY dataTypeSize : UINT
GET
dataTypeSize := SIZEOF(_value);
END_GET
END_PROPERTY

METHOD get_value : BOOL
VAR_OUTPUT
	value : UINT ;
	errId : UDINT;
END_VAR
IF init_done THEN
	value := _value;
	get_value := TRUE;
ELSE
	errId := 2;
	get_value := FALSE;
END_IF
END_METHOD

METHOD handle_read_callback : BOOL
VAR_INPUT
	pt_buffer : POINTER TO CoE_buffer_type_cast_union;
	errId : UDINT;
END_VAR

_value := pt_buffer^.value_uint;
_init_done:=TRUE;
_read_errId:=errId;
END_METHOD

METHOD set_value : BOOL
VAR_INPUT
	value : uint ;
END_VAR
_valueToWrite.value_uint := value;
IF THIS^._I_CoE_communication_handler <> 0 THEN 
	THIS^._I_CoE_communication_handler.add_write_request(THIS^);
ELSE
	errId:=1;
END_IF
END_METHOD

END_FUNCTION_BLOCK

// ---- _internal/CoE/properties/CoE_property_string.TcPOU
FUNCTION_BLOCK CoE_property_string EXTENDS CoE_property
VAR_INPUT
END_VAR
VAR_OUTPUT
END_VAR
VAR
		_value : STRING;
END_VAR

SUPER^();

PROPERTY dataTypeSize : UINT
GET
dataTypeSize := SIZEOF(_value);
END_GET
END_PROPERTY

METHOD get_value : BOOL
VAR_OUTPUT
	value : STRING ;
	errId : UDINT;
END_VAR
IF init_done THEN
	value := _value;
	get_value := TRUE;
ELSE
	errId := 2;
	get_value := FALSE;
END_IF
END_METHOD

METHOD handle_read_callback : BOOL
VAR_INPUT
	pt_buffer : POINTER TO CoE_buffer_type_cast_union;
	errId : UDINT;
END_VAR

_value := pt_buffer^.value_string;
_init_done:=TRUE;
_read_errId:=errId;
END_METHOD

METHOD set_value : BOOL
VAR_INPUT
	value : string ;
END_VAR
_valueToWrite.value_string := value;
IF THIS^._I_CoE_communication_handler <> 0 THEN 
	THIS^._I_CoE_communication_handler.add_write_request(THIS^);
ELSE
	errId:=1;
END_IF
END_METHOD

END_FUNCTION_BLOCK

// ---- _internal/CoE/properties/CoE_property_udint.TcPOU
FUNCTION_BLOCK CoE_property_udint EXTENDS CoE_property
VAR_INPUT
END_VAR
VAR_OUTPUT
END_VAR
VAR
	_value : UDINT;
END_VAR

SUPER^();

PROPERTY dataTypeSize : UINT
GET
dataTypeSize := SIZEOF(_value);
END_GET
END_PROPERTY

METHOD get_value : BOOL
VAR_OUTPUT
	value : UDINT ;
	errId : UDINT;
END_VAR
IF init_done THEN
	value := _value;
	get_value := TRUE;
ELSE
	errId := 2;
	get_value := FALSE;
END_IF
END_METHOD

METHOD handle_read_callback : BOOL
VAR_INPUT
	pt_buffer : POINTER TO CoE_buffer_type_cast_union;
	errId : UDINT;
END_VAR

_value := pt_buffer^.value_udint;
_init_done:=TRUE;
_read_errId:=errId;
END_METHOD

METHOD set_value : BOOL
VAR_INPUT
	value : UDINT ;
END_VAR
_valueToWrite.value_udint := value;
IF THIS^._I_CoE_communication_handler <> 0 THEN 
	THIS^._I_CoE_communication_handler.add_write_request(THIS^);
ELSE
	errId:=1;
END_IF
END_METHOD

END_FUNCTION_BLOCK

